DATA_BLOCK "DB00851_St_ConstAiScaleData"   // DB851
TITLE = Static DB [SYSTEM CONSTANTS] — Analog Input Scale Data and Ranges
{ S7_Optimized_Access := 'TRUE' }
AUTHOR : M_Gledhill
FAMILY : SysConstants
NAME : St_ConstAiScaleData
VERSION : 1.0
// PRACTICAL SERIES AUTOMATION LIBRARY (PAL)   —   COPYRIGHT 2020 – M. GLEDHILL (MIT LICENCE)
//                   ———— ◆ ————
// FULL ONLINE DOCUMENTATION IS AVAILABLE AT: https://practicalseries.com/2001-pal/index.html
// stored: AutoNumber false, DBAccessibleFromOPCUA true, IsOnlyStoredInLoadMemory false, IsRetainMemResEnabled false, IsWriteProtectedInAS false, MemoryReserve 100
   VAR
      _DB_Header { ExternalAccessible := 'False'; ExternalVisible := 'False'; ExternalWritable := 'False'} : Array[0..79] of Bool;   // Static DB [SYSTEM CONSTANTS] — Analog Input Scale Data and Ranges
      __________0000_0 { ExternalAccessible := 'False'; ExternalVisible := 'False'; ExternalWritable := 'False'} : Bool := false;
      __________0000_1 { ExternalAccessible := 'False'; ExternalVisible := 'False'; ExternalWritable := 'False'} : Bool := false;
      revInfo { ExternalWritable := 'False'} : "UT01000_St_SysRevision";
      __________0010_0 { ExternalAccessible := 'False'; ExternalVisible := 'False'; ExternalWritable := 'False'} : Bool := false;
      __________0010_1 { ExternalAccessible := 'False'; ExternalVisible := 'False'; ExternalWritable := 'False'} : Bool := false;   // ▀▀▀▀ ANALOG SCALE SIGNALS — TEST SIGNALS
      AI_SCALE_TST001 { ExternalWritable := 'False'; S7_SetPoint := 'True'} : "UT00851_Sy_ConstAiScaleData";   // Test range — 0 to 1000 l/s
      AI_SCALE_TST002 { ExternalWritable := 'False'; S7_SetPoint := 'True'} : "UT00851_Sy_ConstAiScaleData";   // Test range — -500 to +500 l/s
      AI_SCALE_TST003 { ExternalWritable := 'False'; S7_SetPoint := 'True'} : "UT00851_Sy_ConstAiScaleData";   // Test range — -1000 to 0 l/s
      AI_SCALE_TST004 { ExternalWritable := 'False'; S7_SetPoint := 'True'} : "UT00851_Sy_ConstAiScaleData";   // Test range — -270 to +1372 DegC
      AI_SCALE_TST005 { ExternalWritable := 'False'; S7_SetPoint := 'True'} : "UT00851_Sy_ConstAiScaleData";   // Test range — Erroneous configuration
      __________0020_0 { ExternalAccessible := 'False'; ExternalVisible := 'False'; ExternalWritable := 'False'} : Bool := false;
      __________0020_1 { ExternalAccessible := 'False'; ExternalVisible := 'False'; ExternalWritable := 'False'} : Bool := false;   // ▀▀▀▀ ANALOG SCALE SIGNALS — INSTRUMENTS
      AI_SCALE_TST006 { ExternalWritable := 'False'; S7_SetPoint := 'True'} : "UT00851_Sy_ConstAiScaleData";   // Test range — 0 to 1000 l/s
      AI_SCALE_FIC001 { ExternalWritable := 'False'; S7_SetPoint := 'True'} : "UT00851_Sy_ConstAiScaleData";   // Inlet flow meter (0-100 l/s)
      AI_SCALE_LIC001 { ExternalWritable := 'False'; S7_SetPoint := 'True'} : "UT00851_Sy_ConstAiScaleData";   // Inlet tank level (0-50 m3)
      AI_SCALE_PIC301 { ExternalWritable := 'False'; S7_SetPoint := 'True'} : "UT00851_Sy_ConstAiScaleData";   // Inlet filter differential pressure (0-2 BarG)
      AI_SCALE_PIC302 { ExternalWritable := 'False'; S7_SetPoint := 'True'} : "UT00851_Sy_ConstAiScaleData";   // Inlet filter differential pressure (0-2 BarG)
   END_VAR
BEGIN
   // _DB_Header[0] : ▄▄▄▄▄▄▄▄▄▄▄▄▄▄▄▄▄▄▄▄▄▄▄▄▄▄▄▄▄▄▄▄ ＣＯＮＳＴＡＮＴＳ ▄▄
   // _DB_Header[2] : TITLE: SYSTEM CONSTANTS — ANALOG INPUT SCALE DATA AND RANGES
   // _DB_Header[4] : ▀▀▀▀▀▀▀▀▀▀▀▀▀▀▀▀▀▀▀▀▀▀▀▀▀▀▀▀▀▀▀▀▀▀▀▀▀▀▀▀▀▀▀▀
   // _DB_Header[5] : TYPE: STATIC
   // _DB_Header[6] : ▄▄▄▄▄▄▄▄▄▄▄▄▄▄▄▄▄▄▄▄▄▄▄▄▄▄▄▄▄▄▄▄▄▄▄▄▄▄▄▄ ʷᴵᴰ⁻ᵈʰᵇ ▄
   // _DB_Header[8] : DB00851_St_ConstAiScaleData is a static data block that holds a full set of scaled ranges,
   // _DB_Header[9] : engineering units, device tag and descriptive data for all types of analog input scaled signals.
   // _DB_Header[11] : Each dataset is stored in a structure of user data type: UT00851_St_ConstAiScaleData.
   // _DB_Header[12] : This structure is configured to hold all the data required to name, scale and apply engineering
   // _DB_Header[13] : units to an analog input signal.
   // _DB_Header[15] : The scaled signal data is stored as constants and is used by all modules that have an interface
   // _DB_Header[16] : to an analog input card.
   // _DB_Header[18] : The purpose of the user data type and associated data block is to provide a consistent set of
   // _DB_Header[19] : scaled ranges and other data for each device or instrument that is available to the Controller
   // _DB_Header[20] : as an analog input.
   // _DB_Header[22] : The ranges correspond to the scaled values returned by the instrument or device, for example,
   // _DB_Header[23] : a flow meter may have a scaled range of -50 l/s to 200 l/s.
   // _DB_Header[25] : In addition, each dataset contains the instrument or device tag (e.g. FIC001), the engineering
   // _DB_Header[26] : units in use (e.g. l/s, kg/hour, °C, % &c.), over-range and under-range limits, a textual description
   // _DB_Header[27] : of the function of the instrument or device e.g. inlet flowmeter (0 l/s to 100 l/s) and additional
   // _DB_Header[28] : user specific information.
   // _DB_Header[30] : The PDF version of the SMDS for this module is available online here:
   // _DB_Header[31] : http://psop.uk/pal-smds-db00851-p
   // _DB_Header[33] : ━━━ ⬙⬙⬙⬙⬙⬙ ━━━
   // _DB_Header[35] : ▄▄▄▄▄▄▄▄▄▄▄▄▄▄▄▄▄▄▄▄▄▄▄▄▄▄▄▄▄▄▄▄▄▄▄▄▄▄▄▄▄▄▄▄
   // _DB_Header[36] : MODIFICATION HISTORY
   // _DB_Header[38] : This is a summary of the recent software modifications made to this block (most recent at top)
   // _DB_Header[40] : ―――――――――――――――――――――――――――――――――――――――――――
   // _DB_Header[41] : DATE REVISION MASTER BRANCH DEV
   // _DB_Header[42] : (nnn.amm) COMMIT TAG (Base ---> Merge) BRANCH Author
   // _DB_Header[43] : ———————————————————————————————————————————
   // _DB_Header[44] : 2022.05.15 001.000 D0018 D0017 D0018 None M. Gledhill
   // _DB_Header[45] : DB00851 — RELEASED FOR USE
   // _DB_Header[46] : Merge back to master branch
   // _DB_Header[48] : 2024.05.15 001.000 D0017A-000.104 D0017 N/A D0017A M. Gledhill
   // _DB_Header[49] : DB00851 — RELEASED FOR USE
   // _DB_Header[51] : 2024.05.03 000.801 D0017A-000.102 D0017 N/A D0017A M. Gledhill
   // _DB_Header[52] : DB00851 Block populated
   // _DB_Header[54] : 2024.04.09 000.101 D0017A-000.101 D0017 N/A D0017A M. Gledhill
   // _DB_Header[55] : DB00851 Block created
   // _DB_Header[56] : ———————————————————————————————————————————
   // _DB_Header[57] : Where: nnn = Major revision
   // _DB_Header[58] : a = Type (1-7 Development, 8 Proving, 9 Qualification, 0 Release)
   // _DB_Header[59] : mm = Minor revision (must be 00 if a = 0)
   // _DB_Header[60] : Block properties version number should be set to nn.a (only one decimal place)
   // _DB_Header[62] : ██████████████ █ █ █ █ END █ █ █ █ ██████████████
   revInfo.REV_BLOCK := 'DB00851';
   revInfo.REV_NUMBER := '001.000';
   revInfo.REV_DATE := '2024-05-15';
   revInfo.REV_AUTHOR := 'M. Gledhill';
   AI_SCALE_TST001.AI_TAG := 'TST001';
   AI_SCALE_TST001.SCALE_MIN := 0.0;
   AI_SCALE_TST001.SCALE_MAX := 1000.0;
   AI_SCALE_TST001.SCALE_UNITS := 'l/s';
   AI_SCALE_TST001.SCALE_DESC := 'Test Range (0 to 1000 l/s)';
   AI_SCALE_TST001.LIMIT_UNDER := -62.5;
   AI_SCALE_TST001.LIMIT_OVER := 1062.5;
   AI_SCALE_TST002.AI_TAG := 'TST002';
   AI_SCALE_TST002.SCALE_MIN := -500.0;
   AI_SCALE_TST002.SCALE_MAX := 500.0;
   AI_SCALE_TST002.SCALE_UNITS := 'l/s';
   AI_SCALE_TST002.SCALE_DESC := 'Test Range (-500 to 500 l/s)';
   AI_SCALE_TST002.LIMIT_UNDER := -562.5;
   AI_SCALE_TST002.LIMIT_OVER := 562.5;
   AI_SCALE_TST003.AI_TAG := 'TST003';
   AI_SCALE_TST003.SCALE_MIN := -1000.0;
   AI_SCALE_TST003.SCALE_MAX := 0.0;
   AI_SCALE_TST003.SCALE_UNITS := 'l/s';
   AI_SCALE_TST003.SCALE_DESC := 'Test Range (-1000 to 0 l/s)';
   AI_SCALE_TST003.LIMIT_UNDER := -1062.5;
   AI_SCALE_TST003.LIMIT_OVER := 62.5;
   AI_SCALE_TST004.AI_TAG := 'TST005';
   AI_SCALE_TST004.SCALE_MIN := -270.0;
   AI_SCALE_TST004.SCALE_MAX := 1372.0;
   AI_SCALE_TST004.SCALE_UNITS := 'DegC';
   AI_SCALE_TST004.SCALE_DESC := 'Test Range (-270 to +1372 DegC)';
   AI_SCALE_TST004.LIMIT_UNDER := -300.0;
   AI_SCALE_TST004.LIMIT_OVER := 1400.0;
   AI_SCALE_TST005.AI_TAG := 'TST005';
   AI_SCALE_TST005.___________0020_0 := false;
   AI_SCALE_TST005.___________0020_1 := false;
   AI_SCALE_TST005.SCALE_MIN := 0.0;
   AI_SCALE_TST005.SCALE_MAX := 1000.0;
   AI_SCALE_TST005.SCALE_UNITS := 'l/s';
   AI_SCALE_TST005.SCALE_DESC := 'Test Range (0 to 1000 l/s)';
   AI_SCALE_TST005.___________0030_0 := false;
   AI_SCALE_TST005.___________0030_1 := false;
   AI_SCALE_TST005.LIMIT_UNDER := 100.0;
   AI_SCALE_TST005.LIMIT_OVER := 900.0;
   AI_SCALE_TST006.AI_TAG := 'TST005';
   AI_SCALE_TST006.SCALE_MIN := 0.0;
   AI_SCALE_TST006.SCALE_MAX := 1000.0;
   AI_SCALE_TST006.SCALE_UNITS := 'l/s';
   AI_SCALE_TST006.SCALE_DESC := 'Test Range (0 to 1000 l/s)';
   AI_SCALE_TST006.LIMIT_UNDER := 100.0;
   AI_SCALE_TST006.LIMIT_OVER := 900.0;
   AI_SCALE_FIC001.AI_TAG := 'FIC001';
   AI_SCALE_FIC001.SCALE_MIN := 0.0;
   AI_SCALE_FIC001.SCALE_MAX := 100.0;
   AI_SCALE_FIC001.SCALE_UNITS := 'l/s';
   AI_SCALE_FIC001.SCALE_DESC := 'Inlet flow meter (0-100 l/s)';
   AI_SCALE_FIC001.LIMIT_UNDER := -5.0;
   AI_SCALE_FIC001.LIMIT_OVER := 105.0;
   AI_SCALE_FIC001.USER_INFO_1 := 'Instrument manufacturer: Siemens';
   AI_SCALE_FIC001.USER_INFO_2 := 'Instrument type: Sitrans FM MAG 5000 (mass flow)';
   AI_SCALE_FIC001.USER_INFO_3 := 'Instrument part no.: 7ME5920-1AA10-1AA0';
   AI_SCALE_FIC001.USER_INFO_4 := 'Instrument serial no.: 3443201102';
   AI_SCALE_LIC001.AI_TAG := 'LIC001';
   AI_SCALE_LIC001.SCALE_MIN := 0.0;
   AI_SCALE_LIC001.SCALE_MAX := 50.0;
   AI_SCALE_LIC001.SCALE_UNITS := 'm3';
   AI_SCALE_LIC001.SCALE_DESC := 'Inlet tank level (0-50 m3)';
   AI_SCALE_LIC001.LIMIT_UNDER := -2.5;
   AI_SCALE_LIC001.LIMIT_OVER := 52.5;
   AI_SCALE_LIC001.USER_INFO_1 := 'Instrument manufacturer: Siemens';
   AI_SCALE_LIC001.USER_INFO_2 := 'Instrument type: Sitrans LU240 (level)';
   AI_SCALE_LIC001.USER_INFO_3 := 'Instrument part no.: 7ML5110-1DD07-4AF0';
   AI_SCALE_LIC001.USER_INFO_4 := 'Instrument serial no.: 4514461005';
   AI_SCALE_PIC301.AI_TAG := 'PIC301';
   AI_SCALE_PIC301.SCALE_MIN := 0.0;
   AI_SCALE_PIC301.SCALE_MAX := 2.0;
   AI_SCALE_PIC301.SCALE_UNITS := 'BarG';
   AI_SCALE_PIC301.SCALE_DESC := 'Inlet filter differential pressure (0-2 BarG)';
   AI_SCALE_PIC301.LIMIT_UNDER := -0.1;
   AI_SCALE_PIC301.LIMIT_OVER := 2.1;
   AI_SCALE_PIC301.USER_INFO_1 := 'Instrument manufacturer: Siemens';
   AI_SCALE_PIC301.USER_INFO_2 := 'Instrument type: Sitrans P420 (pressure)';
   AI_SCALE_PIC301.USER_INFO_3 := 'Instrument part no.: 7MF0440-1ML02-5BF0';
   AI_SCALE_PIC301.USER_INFO_4 := 'Instrument serial no.: 7875344001';
   AI_SCALE_PIC302.AI_TAG := 'PIC301';
   AI_SCALE_PIC302.SCALE_MIN := 0.0;
   AI_SCALE_PIC302.SCALE_MAX := 2.0;
   AI_SCALE_PIC302.SCALE_UNITS := 'BarG';
   AI_SCALE_PIC302.SCALE_DESC := 'Inlet filter differential pressure (0-2 BarG)';
   AI_SCALE_PIC302.LIMIT_UNDER := -0.1;
   AI_SCALE_PIC302.LIMIT_OVER := 2.1;
   AI_SCALE_PIC302.USER_INFO_1 := 'Instrument manufacturer: Siemens';
   AI_SCALE_PIC302.USER_INFO_2 := 'Instrument type: Sitrans P420 (pressure)';
   AI_SCALE_PIC302.USER_INFO_3 := 'Instrument part no.: 7MF0440-1ML02-5BF0';
   AI_SCALE_PIC302.USER_INFO_4 := 'Instrument serial no.: 7875344008';
END_DATA_BLOCK

DATA_BLOCK "DB00852_St_ConstAqScaleData"   // DB852
TITLE = Static DB [SYSTEM CONSTANTS] — Analog Input Scale Data and Ranges
{ S7_Optimized_Access := 'TRUE' }
AUTHOR : M_Gledhill
FAMILY : SysConstants
NAME : St_ConstAiScaleData
VERSION : 1.0
// PRACTICAL SERIES AUTOMATION LIBRARY (PAL)   —   COPYRIGHT 2020 – M. GLEDHILL (MIT LICENCE)
//                   ———— ◆ ————
// FULL ONLINE DOCUMENTATION IS AVAILABLE AT: https://practicalseries.com/2001-pal/index.html
// stored: AutoNumber false, DBAccessibleFromOPCUA true, IsOnlyStoredInLoadMemory false, IsRetainMemResEnabled false, IsWriteProtectedInAS false, MemoryReserve 100
   VAR
      _DB_Header { ExternalAccessible := 'False'; ExternalVisible := 'False'; ExternalWritable := 'False'} : Array[0..79] of Bool;   // Static DB [SYSTEM CONSTANTS] — Analog Instrument Scale Data and Ranges
      __________0000_0 { ExternalAccessible := 'False'; ExternalVisible := 'False'; ExternalWritable := 'False'} : Bool := false;
      __________0000_1 { ExternalAccessible := 'False'; ExternalVisible := 'False'; ExternalWritable := 'False'} : Bool := false;
      revInfo { ExternalWritable := 'False'} : "UT01000_St_SysRevision";
      __________0010_0 { ExternalAccessible := 'False'; ExternalVisible := 'False'; ExternalWritable := 'False'} : Bool := false;
      __________0010_1 { ExternalAccessible := 'False'; ExternalVisible := 'False'; ExternalWritable := 'False'} : Bool := false;   // ▀▀▀▀ ANALOG SCALE SIGNALS — MODULATING VALVES
      AQ_SCALE_FCV001_DMD { ExternalWritable := 'False'; S7_SetPoint := 'True'} : "UT00852_Sy_ConstAqScaleData";   // Inlet flow control valve position demand (0 to 100%)
      __________0020_0 { ExternalAccessible := 'False'; ExternalVisible := 'False'; ExternalWritable := 'False'} : Bool := false;
      __________0020_1 { ExternalAccessible := 'False'; ExternalVisible := 'False'; ExternalWritable := 'False'} : Bool := false;   // ▀▀▀▀ ANALOG SCALE SIGNALS — CHART RECORDER
      AQ_SCALE_REC001 { ExternalWritable := 'False'; S7_SetPoint := 'True'} : "UT00852_Sy_ConstAqScaleData";   // Recorder - Inlet flow meter (0-100 l/s)
      AQ_SCALE_REC002 { ExternalWritable := 'False'; S7_SetPoint := 'True'} : "UT00852_Sy_ConstAqScaleData";   // Recorder - Inlet tank level (0-50 m3)
   END_VAR
BEGIN
   // _DB_Header[0] : ▄▄▄▄▄▄▄▄▄▄▄▄▄▄▄▄▄▄▄▄▄▄▄▄▄▄▄▄▄▄▄▄ ＣＯＮＳＴＡＮＴＳ ▄▄
   // _DB_Header[2] : TITLE: SYSTEM CONSTANTS — ANALOG INPUT SCALE DATA AND RANGES
   // _DB_Header[4] : ▀▀▀▀▀▀▀▀▀▀▀▀▀▀▀▀▀▀▀▀▀▀▀▀▀▀▀▀▀▀▀▀▀▀▀▀▀▀▀▀▀▀▀▀
   // _DB_Header[5] : TYPE: STATIC
   // _DB_Header[6] : ▄▄▄▄▄▄▄▄▄▄▄▄▄▄▄▄▄▄▄▄▄▄▄▄▄▄▄▄▄▄▄▄▄▄▄▄▄▄▄▄ ʷᴵᴰ⁻ᵈʰᵇ ▄
   // _DB_Header[8] : DB00852_St_ConstAqScaleData is a static data block that holds a full set of scaled ranges,
   // _DB_Header[9] : engineering units, device tag and descriptive data for all types of analog output scaled signals.
   // _DB_Header[11] : Each dataset is stored in a structure of user data type: UT00852_St_ConstAqScaleData.
   // _DB_Header[12] : This structure is configured to hold all the data required to name, scale and apply engineering
   // _DB_Header[13] : units to an analog output signal.
   // _DB_Header[15] : All the scaled signal data is stored as constants and is used by all modules that have an interface
   // _DB_Header[16] : to an analog output card.
   // _DB_Header[18] : The purpose of the user data type and associated data block is to provide a consistent set of
   // _DB_Header[19] : scaled ranges and other data for each device that is available to the Controller
   // _DB_Header[20] : as an analog output.
   // _DB_Header[22] : The ranges correspond to the scaled values of a signal that is to be converted into an analog
   // _DB_Header[23] : output, for example, a modulating valve may have a scaled range of 0% to 100%.
   // _DB_Header[25] : In addition, each dataset contains the device tag (e.g. FCV001), the engineering
   // _DB_Header[26] : units in use (e.g. l/s, kg/hour, °C, % &c.), over-range and under-range limits, a textual description
   // _DB_Header[27] : of the function of the device e.g.inlet flow control valve and additional user specific
   // _DB_Header[28] : information.
   // _DB_Header[30] : The PDF version of the SMDS for this module is available online here:
   // _DB_Header[31] : http://psop.uk/pal-smds-db00851-p
   // _DB_Header[33] : ━━━ ⬙⬙⬙⬙⬙⬙ ━━━
   // _DB_Header[35] : ▄▄▄▄▄▄▄▄▄▄▄▄▄▄▄▄▄▄▄▄▄▄▄▄▄▄▄▄▄▄▄▄▄▄▄▄▄▄▄▄▄▄▄▄
   // _DB_Header[36] : MODIFICATION HISTORY
   // _DB_Header[38] : This is a summary of the recent software modifications made to this block (most recent at top)
   // _DB_Header[40] : ―――――――――――――――――――――――――――――――――――――――――――
   // _DB_Header[41] : DATE REVISION MASTER BRANCH DEV
   // _DB_Header[42] : (nnn.amm) COMMIT TAG (Base ---> Merge) BRANCH Author
   // _DB_Header[43] : ———————————————————————————————————————————
   // _DB_Header[44] : 2024.05.17 001.000 D0017A-000.104 D0017 N/A D0017A M. Gledhill
   // _DB_Header[45] : DB00852 — RELEASED FOR USE
   // _DB_Header[47] : 2024.05.03 000.801 D0017A-000.102 D0017 N/A D0017A M. Gledhill
   // _DB_Header[48] : DB00852 Block populated
   // _DB_Header[50] : 2024.04.09 000.101 D0017A-000.101 D0017 N/A D0017A M. Gledhill
   // _DB_Header[51] : DB00852 Block created
   // _DB_Header[52] : ———————————————————————————————————————————
   // _DB_Header[53] : Where: nnn = Major revision
   // _DB_Header[54] : a = Type (1-7 Development, 8 Proving, 9 Qualification, 0 Release)
   // _DB_Header[55] : mm = Minor revision (must be 00 if a = 0)
   // _DB_Header[56] : Block properties version number should be set to nn.a (only one decimal place)
   // _DB_Header[58] : ██████████████ █ █ █ █ END █ █ █ █ ██████████████
   revInfo.REV_BLOCK := 'DB00852';
   revInfo.REV_NUMBER := '001.000';
   revInfo.REV_DATE := '2024-05-17';
   revInfo.REV_AUTHOR := 'M. Gledhill';
   AQ_SCALE_FCV001_DMD.AQ_TAG := 'FCV001';
   AQ_SCALE_FCV001_DMD.SCALE_MIN := 0.0;
   AQ_SCALE_FCV001_DMD.SCALE_MAX := 100.0;
   AQ_SCALE_FCV001_DMD.SCALE_UNITS := '%';
   AQ_SCALE_FCV001_DMD.SCALE_DESC := 'Inlet flow control valve (0 to 100%)';
   AQ_SCALE_FCV001_DMD.LIMIT_UNDER := -2.5;
   AQ_SCALE_FCV001_DMD.LIMIT_OVER := 102.5;
   AQ_SCALE_FCV001_DMD.USER_INFO_1 := 'Instrument manufacturer: Siemens';
   AQ_SCALE_FCV001_DMD.USER_INFO_2 := 'Instrument type: 2-port magnetic';
   AQ_SCALE_FCV001_DMD.USER_INFO_3 := 'Instrument part no.: MXG461.15-0.6';
   AQ_SCALE_FCV001_DMD.USER_INFO_4 := 'Instrument serial no.:2075181118';
   AQ_SCALE_REC001.AQ_TAG := 'REC001';
   AQ_SCALE_REC001.SCALE_MIN := 0.0;
   AQ_SCALE_REC001.SCALE_MAX := 100.0;
   AQ_SCALE_REC001.SCALE_UNITS := 'l/s';
   AQ_SCALE_REC001.SCALE_DESC := 'Recorder - Inlet flow meter (0-100 l/s)';
   AQ_SCALE_REC002.AQ_TAG := 'REC002';
   AQ_SCALE_REC002.SCALE_MIN := 0.0;
   AQ_SCALE_REC002.SCALE_MAX := 50.0;
   AQ_SCALE_REC002.SCALE_UNITS := 'm3';
   AQ_SCALE_REC002.SCALE_DESC := 'Recorder - Inlet tank level (0-50 m3)';
END_DATA_BLOCK

DATA_BLOCK "DB21001_Dy_SysGlobalData"   // DB21001
TITLE = Dynamic DB — Sys - Global Data
{ S7_Optimized_Access := 'TRUE' }
AUTHOR : M_Gledhill
FAMILY : System
NAME : Dy_SysGlobalData
VERSION : 1.0
// PRACTICAL SERIES AUTOMATION LIBRARY (PAL)   —   COPYRIGHT 2020 – M. GLEDHILL (MIT LICENCE)
//                   ———— ◆ ————
//  FOR DETAILED DOCUMENTATION — SELECT THE BLOCK IN THE PROJECT TREE AND PRESS SHIFT + F1
//  FULL ONLINE DOCUMENTATION IS AVAILABLE AT: https://practicalseries.com/2001-pal/index.html
// stored: AutoNumber false, DBAccessibleFromOPCUA true, IsOnlyStoredInLoadMemory false, IsRetainMemResEnabled false, IsWriteProtectedInAS false, MemoryReserve 100
   VAR
      _DB_Header { ExternalWritable := 'False'} : Array[0..79] of Bool;   // STANDARD SYSTEM GLOBAL DATA
      __________0000_0 { ExternalWritable := 'False'} : Bool := false;
      __________0000_1 { ExternalWritable := 'False'} : Bool := false;   // ▀▀▀▀ DB CURRENT REVISION
      revInfo { ExternalWritable := 'False'} : "UT01000_St_SysRevision";
      __________0010_0 { ExternalWritable := 'False'} : Bool := false;
      __________0010_1 { ExternalWritable := 'False'} : Bool := false;   // ▀▀▀▀ PROJECT CURRENT REVISION
      projRevInfo { ExternalWritable := 'False'} : "UT01000_St_SysRevision";
      __________0020_0 { ExternalWritable := 'False'} : Bool := false;
      __________0020_1 { ExternalWritable := 'False'} : Bool := false;   // ▀▀▀▀ SYSTEM SIGNALS — LOGIC AND TIMING SIGNALS
      SysSignals { ExternalWritable := 'False'} : "UT21000_Dy_SysSignals";
      __________0030_0 { ExternalWritable := 'False'} : Bool := false;
      __________0030_1 { ExternalWritable := 'False'} : Bool := false;   // ▀▀▀▀ SYSTEM DATA — CYCLE TIMING AND RTC
      SysData { ExternalWritable := 'False'} : "UT21001_Dy_SysData";
      __________0040_0 { ExternalWritable := 'False'} : Bool := false;
      __________0040_1 { ExternalWritable := 'False'} : Bool := false;   // ▀▀▀▀ OB CALL TIMES
      OB10_CallTime { ExternalWritable := 'False'} : DTL;   // Time of day interrupt 1
      OB11_CallTime { ExternalWritable := 'False'} : DTL;   // Time of day interrupt 2
      OB12_CallTime { ExternalWritable := 'False'} : DTL;   // Time of day interrupt 3
      OB13_CallTime { ExternalWritable := 'False'} : DTL;   // Time of day interrupt 4
      OB14_CallTime { ExternalWritable := 'False'} : DTL;   // Time of day interrupt 5
      OB15_CallTime { ExternalWritable := 'False'} : DTL;   // Time of day interrupt 6
      OB16_CallTime { ExternalWritable := 'False'} : DTL;   // Time of day interrupt 7
      OB17_CallTime { ExternalWritable := 'False'} : DTL;   // Time of day interrupt 8
      OB20_CallTime { ExternalWritable := 'False'} : DTL;   // Time delay interrupt 1
      OB21_CallTime { ExternalWritable := 'False'} : DTL;   // Time delay interrupt 2
      OB22_CallTime { ExternalWritable := 'False'} : DTL;   // Time delay interrupt 3
      OB23_CallTime { ExternalWritable := 'False'} : DTL;   // Time delay interrupt 4
      OB30_CallTime { ExternalWritable := 'False'} : DTL;   // Timed cyclic interrupt 1
      OB31_CallTime { ExternalWritable := 'False'} : DTL;   // Timed cyclic interrupt 2
      OB32_CallTime { ExternalWritable := 'False'} : DTL;   // Timed cyclic interrupt 3
      OB33_CallTime { ExternalWritable := 'False'} : DTL;   // Timed cyclic interrupt 4
      OB34_CallTime { ExternalWritable := 'False'} : DTL;   // Timed cyclic interrupt 5
      OB35_CallTime { ExternalWritable := 'False'} : DTL;   // Timed cyclic interrupt 6
      OB36_CallTime { ExternalWritable := 'False'} : DTL;   // Timed cyclic interrupt 7
      OB37_CallTime { ExternalWritable := 'False'} : DTL;   // Timed cyclic interrupt 8
      OB38_CallTime { ExternalWritable := 'False'} : DTL;   // Timed cyclic interrupt 9
      OB40_CallTime { ExternalWritable := 'False'} : DTL;   // Hardware interrupt 1
      OB41_CallTime { ExternalWritable := 'False'} : DTL;   // Hardware interrupt 2
      OB42_CallTime { ExternalWritable := 'False'} : DTL;   // Hardware interrupt 3
      OB43_CallTime { ExternalWritable := 'False'} : DTL;   // Hardware interrupt 4
      OB44_CallTime { ExternalWritable := 'False'} : DTL;   // Hardware interrupt 5
      OB45_CallTime { ExternalWritable := 'False'} : DTL;   // Hardware interrupt 6
      OB46_CallTime { ExternalWritable := 'False'} : DTL;   // Hardware interrupt 7
      OB47_CallTime { ExternalWritable := 'False'} : DTL;   // Hardware interrupt 8
      OB80_CallTime { ExternalWritable := 'False'} : DTL;   // Error interrupt — max cycle time exceeded
      OB82_CallTime { ExternalWritable := 'False'} : DTL;   // Error interrupt — module diagnostic
      OB83_CallTime { ExternalWritable := 'False'} : DTL;   // Error interrupt — module changed
      OB86_CallTime { ExternalWritable := 'False'} : DTL;   // Error interrupt — rack fault
      OB100_CallTime { ExternalWritable := 'False'} : DTL;   // Start-up interrupt
      OB121_CallTime { ExternalWritable := 'False'} : DTL;   // Error interrupt — programming fault
      OB122_CallTime { ExternalWritable := 'False'} : DTL;   // Error interrupt — IO access fault
   END_VAR
BEGIN
   // _DB_Header[0] : ▀▀▀▀▀▀▀▀▀▀▀▀▀▀▀▀▀▀▀▀▀▀▀▀▀▀▀▀▀▀▀▀▀▀▀▀▀▀▀▀▀▀▀▀
   // _DB_Header[2] : TITLE: STANDARD SYSTEM GLOBAL DATA
   // _DB_Header[4] : ▄▄▄▄▄▄▄▄▄▄▄▄▄▄▄▄▄▄▄▄▄▄▄▄▄▄▄▄▄▄▄▄▄▄▄▄▄▄▄▄▄▄▄▄
   // _DB_Header[5] : TYPE: DYNAMIC
   // _DB_Header[6] : ▀▀▀▀▀▀▀▀▀▀▀▀▀▀▀▀▀▀▀▀▀▀▀▀▀▀▀▀▀▀▀▀▀▀▀▀▀▀▀▀▀▀▀▀
   // _DB_Header[8] : Global system data storage DB. The block records various system variables and information:
   // _DB_Header[10] : • Project revision data
   // _DB_Header[11] : • Common system signals (logic and timing)
   // _DB_Header[12] : • Cycle timing information (previous, max, min and a cycle counter)
   // _DB_Header[13] : • CPU real time clock data (in globally readable format)
   // _DB_Header[14] : • Last call time of any interrupt OB
   // _DB_Header[16] : The cycle timing information and the RTC data are provided by FC01000. The interrupt OB data
   // _DB_Header[17] : is provided by the individual OBs.
   // _DB_Header[19] : ━━━ ⬙⬙⬙⬙⬙⬙ ━━━
   // _DB_Header[21] : ▄▄▄▄▄▄▄▄▄▄▄▄▄▄▄▄▄▄▄▄▄▄▄▄▄▄▄▄▄▄▄▄▄▄▄▄▄▄▄▄▄▄▄▄
   // _DB_Header[22] : MODIFICATION HISTORY
   // _DB_Header[24] : This is a summary of the recent software modifications made to this block (most recent at top)
   // _DB_Header[26] : ―――――――――――――――――――――――――――――――――――――――――――
   // _DB_Header[27] : DATE REVISION MASTER BRANCH DEV
   // _DB_Header[28] : (nnn.amm) COMMIT TAG (Base ---> Merge) BRANCH Author
   // _DB_Header[29] : ———————————————————————————————————————————
   // _DB_Header[30] : 2021.05.11 001.000 D0006 D0005 D0006 None M. Gledhill
   // _DB_Header[31] : FC01001 — RELEASED FOR USE
   // _DB_Header[32] : Merge back to master branch
   // _DB_Header[34] : 2021.05.11 000.801 D0005A-000.801 D0005 N/A D0005A M. Gledhill
   // _DB_Header[35] : FC01001 — Released for SMT
   // _DB_Header[37] : 2021.05.08 000.101 D0005A-000.101 D0005 N/A D0005A M. Gledhill
   // _DB_Header[38] : FC01001 Migration to VCS
   // _DB_Header[39] : ———————————————————————————————————————————
   // _DB_Header[41] : ██████████████ █ █ █ █ END █ █ █ █ ██████████████
   revInfo.REV_BLOCK := 'DB21001';
   revInfo.REV_NUMBER := '001.000';
   revInfo.REV_DATE := '2021-05-11';
   revInfo.REV_AUTHOR := 'M. Gledhill';
END_DATA_BLOCK

DATA_BLOCK "DB02001_St_InstAnalogRead"   // DB2001
TITLE = Static DB — Inst - Analog Instrument Read, Scale and Monitor
{ S7_Optimized_Access := 'TRUE' }
AUTHOR : M_Gledhill
FAMILY : Instrumentation
NAME : St_InstAnalogRead
VERSION : 0.1
// PRACTICAL SERIES AUTOMATION LIBRARY (PAL)   —   COPYRIGHT 2020 – M. GLEDHILL (MIT LICENCE)
//                   ———— ◆ ————
//  FOR DETAILED DOCUMENTATION — SELECT THE BLOCK IN THE PROJECT TREE AND PRESS SHIFT + F1
//  FULL ONLINE DOCUMENTATION IS AVAILABLE AT: https://practicalseries.com/2001-pal/index.html
// stored: AutoNumber false, DBAccessibleFromOPCUA true, IsOnlyStoredInLoadMemory false, IsRetainMemResEnabled false, IsWriteProtectedInAS false, MemoryReserve 100
   VAR
      _DB_Header { ExternalAccessible := 'False'; ExternalVisible := 'False'; ExternalWritable := 'False'} : Array[0..79] of Bool;   // STANDARD ANALOG INSTRUMENT READ
      __________0000_0 { ExternalAccessible := 'False'; ExternalVisible := 'False'; ExternalWritable := 'False'} : Bool := false;
      __________0000_1 { ExternalAccessible := 'False'; ExternalVisible := 'False'; ExternalWritable := 'False'} : Bool := false;   // ▀▀▀▀ DB CURRENT REVISION
      revInfo { ExternalWritable := 'False'; S7_SetPoint := 'True'} : "UT01000_St_SysRevision";
      __________0010_0 { ExternalAccessible := 'False'; ExternalVisible := 'False'; ExternalWritable := 'False'} : Bool := false;
      __________0010_1 { ExternalAccessible := 'False'; ExternalVisible := 'False'; ExternalWritable := 'False'} : Bool := false;   // ▀▀▀▀ ANALOG INSTRUMENTS
      FIC101 { ExternalWritable := 'False'; S7_SetPoint := 'True'} : "UT02001_St_InstAnalogRead";   // Filter 1 outlet flow
   END_VAR
BEGIN
   // _DB_Header[0] : ▀▀▀▀▀▀▀▀▀▀▀▀▀▀▀▀▀▀▀▀▀▀▀▀▀▀▀▀▀▀▀▀▀▀▀▀▀▀▀▀▀▀▀▀
   // _DB_Header[2] : TITLE: STANDARD ANALOG INSTRUMENT READ (SCALE & ALARM MONITORING)
   // _DB_Header[4] : ▄▄▄▄▄▄▄▄▄▄▄▄▄▄▄▄▄▄▄▄▄▄▄▄▄▄▄▄▄▄▄▄▄▄▄▄▄▄▄▄▄▄▄▄
   // _DB_Header[5] : TYPE: STATIC
   // _DB_Header[6] : ▀▀▀▀▀▀▀▀▀▀▀▀▀▀▀▀▀▀▀▀▀▀▀▀▀▀▀▀▀▀▀▀▀▀▀▀▀▀▀▀▀▀▀▀
   // _DB_Header[8] : This is the static data block associated with the standard analog instrument read
   // _DB_Header[9] : block:
   // _DB_Header[10] : FC02001_StdInstAnalogRead
   // _DB_Header[12] : The static data holds the threshold values for any configured alarms and warnings,
   // _DB_Header[13] : activation delays, scaled and raw value ranges and various configuration options.
   // _DB_Header[15] : Each instrument is given the user data type:
   // _DB_Header[16] : UT02001_St_InstAnalogRead
   // _DB_Header[17] : This holds the full set of static configuration data for the instrument.
   // _DB_Header[19] : ━━━ ⬙⬙⬙⬙⬙⬙ ━━━
   // _DB_Header[21] : ▄▄▄▄▄▄▄▄▄▄▄▄▄▄▄▄▄▄▄▄▄▄▄▄▄▄▄▄▄▄▄▄▄▄▄▄▄▄▄▄▄▄▄▄
   // _DB_Header[22] : MODIFICATION HISTORY
   // _DB_Header[24] : This is a summary of the recent software modifications made to this block (most recent at top)
   // _DB_Header[26] : ―――――――――――――――――――――――――――――――――――――――――――
   // _DB_Header[27] : DATE REVISION MASTER BRANCH DEV
   // _DB_Header[28] : (nnn.amm) COMMIT TAG (Base ---> Merge) BRANCH Author
   // _DB_Header[29] : ———————————————————————————————————————————
   // _DB_Header[30] : 2021.05.18 000.101 D0006B-000.101 D0006 N/A D0006B M. Gledhill
   // _DB_Header[31] : FC02001 Migration to VCS
   // _DB_Header[32] : ———————————————————————————————————————————
   // _DB_Header[33] : Where: nnn = Major revision
   // _DB_Header[34] : a = Type (1-7 Development, 8 Proving, 9 Qualification, 0 Release)
   // _DB_Header[35] : mm = Minor revision (must be 00 if a = 0)
   // _DB_Header[36] : Block properties version number should be set to nn.a (only one decimal place)
   // _DB_Header[38] : ██████████████ █ █ █ █ END █ █ █ █ ██████████████
   revInfo.REV_BLOCK := 'DB02001';
   revInfo.REV_NUMBER := '000.101';
   revInfo.REV_DATE := '2021-05-18';
   revInfo.REV_AUTHOR := 'M. Gledhill';
   FIC101.CONFIG_ALM_H_ENABLE := true;
   FIC101.CONFIG_ALM_L_ENABLE := true;
   FIC101.CONFIG_WRN_H_ENABLE := true;
   FIC101.CONFIG_WRN_L_ENABLE := true;
   FIC101.CONFIG_FP_DISABLE := false;
   FIC101.CONFIG_SIM_DISABLE := false;
   FIC101.CONFIG_RL_ENABLE := false;
   FIC101.RANGE_RAW_MAX := 27648;
   FIC101.RANGE_SCALE_MIN := 0.0;
   FIC101.RANGE_SCALE_MAX := 1000.0;
   FIC101.RANGE_OOR_PERCENT := 2.5;
   FIC101.INFO_TAG := 'FIC101';
   FIC101.INFO_UNITS := 'l/s';
   FIC101.SP_ALM_H_VAL := 750.0;
   FIC101.SP_ALM_L_VAL := 250.0;
   FIC101.SP_WRN_H_VAL := 625.0;
   FIC101.SP_WRN_L_VAL := 375.0;
   FIC101.SP_ALM_H_HYST_VAL := 62.5;
   FIC101.SP_ALM_L_HYST_VAL := 62.0;
   FIC101.SP_WRN_H_HYST_VAL := 61.5;
   FIC101.SP_WRN_L_HYST_VAL := 61.0;
   FIC101.TIME_ALM_H_ON_DEL := 10.0;
   FIC101.TIME_ALM_L_ON_DEL := 11.0;
   FIC101.TIME_WRN_H_ON_DEL := 12.0;
   FIC101.TIME_WRN_L_ON_DEL := 13.0;
   FIC101.TIME_ALM_H_OFF_DEL := 15.0;
   FIC101.TIME_ALM_L_OFF_DEL := 16.0;
   FIC101.TIME_WRN_H_OFF_DEL := 17.0;
   FIC101.TIME_WRN_L_OFF_DEL := 18.0;
END_DATA_BLOCK

DATA_BLOCK "DB22001_Dy_InstAnalogRead"   // DB22001
TITLE = Dynamic DB [INSTRUMENTATION] — Analog Instrument Read, Scale and Monitor
{ S7_Optimized_Access := 'TRUE' }
AUTHOR : M_Gledhill
FAMILY : Instrumentation
NAME : Dy_InstAnalogRead
VERSION : 3.0
// PRACTICAL SERIES AUTOMATION LIBRARY (PAL)   —   COPYRIGHT 2020 – M. GLEDHILL (MIT LICENCE)
//                   ———— ◆ ————
// FULL ONLINE DOCUMENTATION IS AVAILABLE AT: https://practicalseries.com/2001-pal/index.html
// stored: AutoNumber false, DBAccessibleFromOPCUA true, IsOnlyStoredInLoadMemory false, IsRetainMemResEnabled false, IsWriteProtectedInAS false, MemoryReserve 100
   VAR
      _DB_Header { ExternalAccessible := 'False'; ExternalVisible := 'False'; ExternalWritable := 'False'} : Array[0..79] of Bool;   // Dynamic DB [INSTRUMENTATION] — Analog Instrument Read, Scale and Monitor
      __________0000_0 { ExternalAccessible := 'False'; ExternalVisible := 'False'; ExternalWritable := 'False'} : Bool := false;
      __________0000_1 { ExternalAccessible := 'False'; ExternalVisible := 'False'; ExternalWritable := 'False'} : Bool := false;   // ▀▀▀▀ DB CURRENT REVISION
      revInfo { ExternalWritable := 'False'; S7_SetPoint := 'True'} : "UT01000_St_SysRevision";   // Revision information
      __________0010_0 { ExternalAccessible := 'False'; ExternalVisible := 'False'; ExternalWritable := 'False'} : Bool := false;
      __________0010_1 { ExternalAccessible := 'False'; ExternalVisible := 'False'; ExternalWritable := 'False'} : Bool := false;   // ▀▀▀▀ ANALOG INSTRUMENTS
      FIC101 { S7_SetPoint := 'True'} : "UT22001_Dy_InstAnalogRead";   // Filter 1 outlet flow
   END_VAR
BEGIN
   // _DB_Header[0] : ▄▄▄▄▄▄▄▄▄▄▄▄▄▄▄▄▄▄▄▄▄▄▄▄▄▄▄▄▄▄▄▄▄ ＳＴＡＮＤＡＲＤ ▄▄
   // _DB_Header[2] : TITLE: INSTRUMENTATION — ANALOG INSTRUMENT READ, SCALE AND MONITOR
   // _DB_Header[4] : ▀▀▀▀▀▀▀▀▀▀▀▀▀▀▀▀▀▀▀▀▀▀▀▀▀▀▀▀▀▀▀▀▀▀▀▀▀▀▀▀▀▀▀▀
   // _DB_Header[5] : TYPE: DYNAMIC
   // _DB_Header[6] : ▄▄▄▄▄▄▄▄▄▄▄▄▄▄▄▄▄▄▄▄▄▄▄▄▄▄▄▄▄▄▄▄▄▄▄▄▄▄▄▄▄▄▄▄
   // _DB_Header[8] : This is the dynamic data block associated with the standard analog instrument read
   // _DB_Header[9] : block:
   // _DB_Header[10] : FC02001_StdInstAnalog
   // _DB_Header[12] : The dynamic data holds the current scaled value of the instrument, along with
   // _DB_Header[13] : any alarms, warnings or faults.
   // _DB_Header[15] : Each instrument is given the user data type:
   // _DB_Header[16] : UT22001_Dy_InstAnalog
   // _DB_Header[17] : This holds the full set of static configuration data for the instrument.
   // _DB_Header[19] : ━━━ ⬙⬙⬙⬙⬙⬙ ━━━
   // _DB_Header[21] : ▄▄▄▄▄▄▄▄▄▄▄▄▄▄▄▄▄▄▄▄▄▄▄▄▄▄▄▄▄▄▄▄▄▄▄▄▄▄▄▄▄▄▄▄
   // _DB_Header[22] : MODIFICATION HISTORY
   // _DB_Header[24] : This is a summary of the recent software modifications made to this block (most recent at top)
   // _DB_Header[26] : ―――――――――――――――――――――――――――――――――――――――――――
   // _DB_Header[27] : DATE REVISION MASTER BRANCH DEV
   // _DB_Header[28] : (nnn.amm) COMMIT TAG (Base ---> Merge) BRANCH Author
   // _DB_Header[29] : ———————————————————————————————————————————
   // _DB_Header[30] : 2024.05.16 003.000 D0017A-000.105 D0017 D0018 None M. Gledhill
   // _DB_Header[31] : FC02001 — RELEASED FOR USE
   // _DB_Header[32] : Merge back to master branch
   // _DB_Header[34] : 2024.05.11 002.801 D0017A-000.104 D0017 N/A D017A M. Gledhill
   // _DB_Header[35] : RAW_ANALOG changed to AI_RAW_SIGNAL
   // _DB_Header[36] : AI_RAW_DATA and AI_SCALE_DATA added and
   // _DB_Header[37] : copied to DYNAMIC_DATA (see db00801 SMDS)
   // _DB_Header[39] : 2022.04.16 002.000 D0011 D0010 D0011 None M. Gledhill
   // _DB_Header[40] : FC02001 — RELEASED FOR USE
   // _DB_Header[41] : Merge back to master branch
   // _DB_Header[43] : 2022.04.11 001.801 D0010A-000.801 D0010 N/A D010A M. Gledhill
   // _DB_Header[44] : Released for test (SCV)
   // _DB_Header[46] : 2022.04.08 001.102 D0010A-000.104 D0010 N/A D010A M. Gledhill
   // _DB_Header[47] : Comments updated
   // _DB_Header[49] : 2022.04.05 001.101 D0010A-000.103 D0010 N/A D010A M. Gledhill
   // _DB_Header[50] : Over and under range based on scaled signal
   // _DB_Header[51] : INFO_TYPE, cal_OR_Abs and cal_UR_Abs added
   // _DB_Header[52] : Comments updated and standardised
   // _DB_Header[53] : UDT variable names standardised
   // _DB_Header[55] : 2021.05.26 001.000 D0008 D0006 D0008 None M. Gledhill
   // _DB_Header[56] : FC02001 — RELEASED FOR USE
   // _DB_Header[57] : Merge back to master branch
   // _DB_Header[59] : 2021.05.24 000.801 D0006B-000.801 D0006 N/A D0006B M. Gledhill
   // _DB_Header[60] : FC02001 — Released for SMT
   // _DB_Header[62] : 2021.05.18 000.101 D0006B-000.101 D0006 N/A D0006B M. Gledhill
   // _DB_Header[63] : FC02001 Migration to VCS
   // _DB_Header[64] : ———————————————————————————————————————————
   // _DB_Header[65] : Where: nnn = Major revision
   // _DB_Header[66] : a = Type (1-7 Development, 8 Proving, 9 Qualification, 0 Release)
   // _DB_Header[67] : mm = Minor revision (must be 00 if a = 0)
   // _DB_Header[68] : Block properties version number should be set to nn.a (only one decimal place)
   // _DB_Header[70] : ██████████████ █ █ █ █ END █ █ █ █ ██████████████
   revInfo.REV_BLOCK := 'DB22001';
   revInfo.REV_NUMBER := '003.000';
   revInfo.REV_DATE := '2024-05-16';
   revInfo.REV_AUTHOR := 'M. Gledhill';
   FIC101.revInfo.REV_BLOCK := 'DB22001';
   FIC101.revInfo.REV_NUMBER := '000.801';
   FIC101.revInfo.REV_DATE := '2021-05-24';
   FIC101.revInfo.REV_AUTHOR := 'M. Gledhill';
END_DATA_BLOCK

DATA_BLOCK "DB11001_St_DevValveIsol"   // DB11001
TITLE = Static DB [Device Driver] — Isolating Valve
{ S7_Optimized_Access := 'TRUE' }
AUTHOR : M_Gledhill
FAMILY : DeviceDriver
NAME : St_StdDevValveIsol
VERSION : 1.0
// PRACTICAL SERIES AUTOMATION LIBRARY (PAL)   —   COPYRIGHT 2020 – M. GLEDHILL (MIT LICENCE)
//                   ———— ◆ ————
//  FOR DETAILED DOCUMENTATION — SELECT THE BLOCK IN THE PROJECT TREE AND PRESS SHIFT + F1
//  FULL ONLINE DOCUMENTATION IS AVAILABLE AT: https://practicalseries.com/2001-pal/index.html
// stored: AutoNumber false, DBAccessibleFromOPCUA true, IsOnlyStoredInLoadMemory false, IsRetainMemResEnabled false, IsWriteProtectedInAS false, MemoryReserve 100
   VAR
      _DB_Header { ExternalAccessible := 'False'; ExternalVisible := 'False'; ExternalWritable := 'False'} : Array[0..79] of Bool;   // STANDARD ANALOG INSTRUMENT READ
      __________0000_0 { ExternalAccessible := 'False'; ExternalVisible := 'False'; ExternalWritable := 'False'} : Bool := false;
      __________0000_1 { ExternalAccessible := 'False'; ExternalVisible := 'False'; ExternalWritable := 'False'} : Bool := false;   // ▀▀▀▀ DB CURRENT REVISION
      revInfo { ExternalWritable := 'False'; S7_SetPoint := 'True'} : "UT01000_St_SysRevision";
      __________0010_0 { ExternalAccessible := 'False'; ExternalVisible := 'False'; ExternalWritable := 'False'} : Bool := false;
      __________0010_1 { ExternalAccessible := 'False'; ExternalVisible := 'False'; ExternalWritable := 'False'} : Bool := false;   // ▀▀▀▀ ISOLATING VALVES
      V001 { ExternalWritable := 'False'} : "UT11001_St_DevValveIsol";   // Filter 1 backwash inlet
   END_VAR
BEGIN
   // _DB_Header[0] : ▀▀▀▀▀▀▀▀▀▀▀▀▀▀▀▀▀▀▀▀▀▀▀▀▀▀▀▀▀▀▀▀▀▀▀▀▀▀▀▀▀▀▀▀
   // _DB_Header[2] : TITLE: STANDARD — DEVICE DRIVER FOR AN ISOLATING VALVE
   // _DB_Header[4] : ▄▄▄▄▄▄▄▄▄▄▄▄▄▄▄▄▄▄▄▄▄▄▄▄▄▄▄▄▄▄▄▄▄▄▄▄▄▄▄▄▄▄▄▄
   // _DB_Header[5] : TYPE: STATIC
   // _DB_Header[6] : ▀▀▀▀▀▀▀▀▀▀▀▀▀▀▀▀▀▀▀▀▀▀▀▀▀▀▀▀▀▀▀▀▀▀▀▀▀▀▀▀▀▀▀▀
   // _DB_Header[8] : This is the static data block associated with the standard device driver for an isolating valve
   // _DB_Header[9] : block:
   // _DB_Header[10] : FC11001_StdDevValveIsol
   // _DB_Header[12] : The static data holds the configuration data for the device (normally open/closed,
   // _DB_Header[13] : limit switch and interlock configuration &c.)
   // _DB_Header[15] : Each instrument is given the user data type:
   // _DB_Header[16] : UT11001_St_DevValveIsol
   // _DB_Header[17] : This holds the full set of static configuration data for the device
   // _DB_Header[19] : ━━━ ⬙⬙⬙⬙⬙⬙ ━━━
   // _DB_Header[21] : ▄▄▄▄▄▄▄▄▄▄▄▄▄▄▄▄▄▄▄▄▄▄▄▄▄▄▄▄▄▄▄▄▄▄▄▄▄▄▄▄▄▄▄▄
   // _DB_Header[22] : MODIFICATION HISTORY
   // _DB_Header[24] : This is a summary of the recent software modifications made to this block (most recent at top)
   // _DB_Header[26] : ―――――――――――――――――――――――――――――――――――――――――――
   // _DB_Header[27] : DATE REVISION MASTER BRANCH DEV
   // _DB_Header[28] : (nnn.amm) COMMIT TAG (Base ---> Merge) BRANCH Author
   // _DB_Header[29] : ———————————————————————————————————————————
   // _DB_Header[30] : 2021.08.23 001.000 D0009 D0008 D0009 None M. Gledhill
   // _DB_Header[31] : FC11001 — RELEASED FOR USE
   // _DB_Header[32] : Merge back to master branch
   // _DB_Header[34] : 2021.08.17 000.801 D0008A-000.801 D0008 N/A D0008A M. Gledhill
   // _DB_Header[35] : FC11001 Released for SMT
   // _DB_Header[37] : 2021.08.10 000.103 D0008A-000.103 D0008 N/A D0008A M. Gledhill
   // _DB_Header[38] : FC11001 Incremental build
   // _DB_Header[40] : 2021.07.21 000.102 D0008A-000.102 D0008 N/A D0008A M. Gledhill
   // _DB_Header[41] : FC11001 Incremental build
   // _DB_Header[43] : 2021.07.08 000.101 D0008A-000.101 D0008 N/A D0008A M. Gledhill
   // _DB_Header[44] : FC11001 Block created
   // _DB_Header[45] : ———————————————————————————————————————————
   // _DB_Header[46] : Where: nnn = Major revision
   // _DB_Header[47] : a = Type (1-7 Development, 8 Proving, 9 Qualification, 0 Release)
   // _DB_Header[48] : mm = Minor revision (must be 00 if a = 0)
   // _DB_Header[49] : Block properties version number should be set to nn.a (only one decimal place)
   // _DB_Header[51] : ██████████████ █ █ █ █ END █ █ █ █ ██████████████
   revInfo.REV_BLOCK := 'DB11001';
   revInfo.REV_NUMBER := '001.000';
   revInfo.REV_DATE := '2021.08.23';
   revInfo.REV_AUTHOR := 'M. Gledhill';
   V001.CONFIG_FBK_OPEN_EN := true;
   V001.CONFIG_FBK_CLOSED_EN := true;
   V001.TIME_OPENING_MAX := 20.0;
   V001.TIME_CLOSING_MAX := 30.0;
   V001.TIME_DER_OPEN := 80.0;
   V001.TIME_DER_CLOSED := 90.0;
END_DATA_BLOCK

DATA_BLOCK "DB11011_St_DevValve3Way"   // DB11011
TITLE = Static DB [DEVICE DRIVER] — Three-Way Valve
{ S7_Optimized_Access := 'TRUE' }
AUTHOR : M_Gledhill
FAMILY : DeviceDriver
NAME : St_DevValve3Way
VERSION : 0.8
// PRACTICAL SERIES AUTOMATION LIBRARY (PAL)   —   COPYRIGHT 2020 – M. GLEDHILL (MIT LICENCE)
//                   ———— ◆ ————
// FULL ONLINE DOCUMENTATION IS AVAILABLE AT: https://practicalseries.com/2001-pal/index.html
// stored: AutoNumber false, DBAccessibleFromOPCUA true, IsOnlyStoredInLoadMemory false, IsRetainMemResEnabled false, IsWriteProtectedInAS false, MemoryReserve 100
   VAR
      _DB_Header { ExternalAccessible := 'False'; ExternalVisible := 'False'; ExternalWritable := 'False'} : Array[0..79] of Bool;   // Static DB [DEVICE DRIVER] — Three-way Valve
      __________0000_0 { ExternalAccessible := 'False'; ExternalVisible := 'False'; ExternalWritable := 'False'} : Bool := false;
      __________0000_1 { ExternalAccessible := 'False'; ExternalVisible := 'False'; ExternalWritable := 'False'} : Bool := false;   // ▀▀▀▀ DB CURRENT REVISION
      revInfo { ExternalWritable := 'False'; S7_SetPoint := 'True'} : "UT01000_St_SysRevision";   // Revision information
      __________0010_0 { ExternalAccessible := 'False'; ExternalVisible := 'False'; ExternalWritable := 'False'} : Bool := false;
      __________0010_1 { ExternalAccessible := 'False'; ExternalVisible := 'False'; ExternalWritable := 'False'} : Bool := false;   // ▀▀▀▀ THREE-WAY VALVES
      V001 { ExternalWritable := 'False'; S7_SetPoint := 'True'} : "UT11011_St_DevValve3Way";   // Filter 1 backwash divert
   END_VAR
BEGIN
   // _DB_Header[0] : ▄▄▄▄▄▄▄▄▄▄▄▄▄▄▄▄▄▄▄▄▄▄▄▄▄▄▄▄▄▄▄▄▄ ＳＴＡＮＤＡＲＤ ▄▄
   // _DB_Header[2] : TITLE: DEVICE DRIVER — THREE-WAY VALVE
   // _DB_Header[4] : ▀▀▀▀▀▀▀▀▀▀▀▀▀▀▀▀▀▀▀▀▀▀▀▀▀▀▀▀▀▀▀▀▀▀▀▀▀▀▀▀▀▀▀▀
   // _DB_Header[5] : TYPE: STATIC
   // _DB_Header[6] : ▄▄▄▄▄▄▄▄▄▄▄▄▄▄▄▄▄▄▄▄▄▄▄▄▄▄▄▄▄▄▄▄▄▄▄▄▄▄▄▄▄▄▄▄
   // _DB_Header[8] : This is the static data block associated with the standard device driver for a three-way valve
   // _DB_Header[9] : block:
   // _DB_Header[10] : FC11011_StdDevValve3Way
   // _DB_Header[12] : The static data holds the configuration data for the device ( limit switch and
   // _DB_Header[13] : interlock configuration &c.)
   // _DB_Header[15] : Each valve is given the user data type:
   // _DB_Header[16] : UT11011_St_DevValve3Way
   // _DB_Header[17] : This holds the full set of static configuration data for the device
   // _DB_Header[19] : ━━━ ⬙⬙⬙⬙⬙⬙ ━━━
   // _DB_Header[21] : ▄▄▄▄▄▄▄▄▄▄▄▄▄▄▄▄▄▄▄▄▄▄▄▄▄▄▄▄▄▄▄▄▄▄▄▄▄▄▄▄▄▄▄▄
   // _DB_Header[22] : MODIFICATION HISTORY
   // _DB_Header[24] : This is a summary of the recent software modifications made to this block (most recent at top)
   // _DB_Header[26] : ―――――――――――――――――――――――――――――――――――――――――――
   // _DB_Header[27] : DATE REVISION MASTER BRANCH DEV
   // _DB_Header[28] : (nnn.amm) COMMIT TAG (Base ---> Merge) BRANCH Author
   // _DB_Header[29] : ———————————————————————————————————————————
   // _DB_Header[30] : 2022.06.07 000.801 D0014A-000.801 D0014 N/A D0014A M. Gledhill
   // _DB_Header[31] : Released for test (SMTS)
   // _DB_Header[33] : 2022.06.01 000.101 D0014A-000.101 D0014 N/A D0014A M. Gledhill
   // _DB_Header[34] : FC11011 Block created
   // _DB_Header[35] : ———————————————————————————————————————————
   // _DB_Header[36] : Where: nnn = Major revision
   // _DB_Header[37] : a = Type (1-7 Development, 8 Proving, 9 Qualification, 0 Release)
   // _DB_Header[38] : mm = Minor revision (must be 00 if a = 0)
   // _DB_Header[39] : Block properties version number should be set to nn.a (only one decimal place)
   // _DB_Header[41] : ██████████████ █ █ █ █ END █ █ █ █ ██████████████
   revInfo.REV_BLOCK := 'DB11011';
   revInfo.REV_NUMBER := '000.801';
   revInfo.REV_DATE := '2022.06.07';
   revInfo.REV_AUTHOR := 'M. Gledhill';
   V001.CONFIG_FBK_ENG_EN := true;
   V001.CONFIG_FBK_DENG_EN := true;
   V001.INFO_TAG := 'V001';
   V001.TIME_ENG_MAX := 20.0;
   V001.TIME_DENG_MAX := 30.0;
   V001.TIME_DER_ENG := 80.0;
   V001.TIME_DER_DENG := 90.0;
END_DATA_BLOCK

DATA_BLOCK "DB11101_St_DevValveBi"   // DB11101
TITLE = Static DB [DEVICE DRIVER] — Bistable Valve
{ S7_Optimized_Access := 'TRUE' }
AUTHOR : M_Gledhill
FAMILY : DeviceDriver
NAME : St_DevValveBi
VERSION : 0.8
// PRACTICAL SERIES AUTOMATION LIBRARY (PAL)   —   COPYRIGHT 2020 – M. GLEDHILL (MIT LICENCE)
//                   ———— ◆ ————
// FULL ONLINE DOCUMENTATION IS AVAILABLE AT: https://practicalseries.com/2001-pal/index.html
// stored: AutoNumber false, DBAccessibleFromOPCUA true, IsOnlyStoredInLoadMemory false, IsRetainMemResEnabled false, IsWriteProtectedInAS false, MemoryReserve 100
   VAR
      _DB_Header { ExternalAccessible := 'False'; ExternalVisible := 'False'; ExternalWritable := 'False'} : Array[0..79] of Bool;   // Static DB [DEVICE DRIVER] — Bistable Valve
      __________0000_0 { ExternalAccessible := 'False'; ExternalVisible := 'False'; ExternalWritable := 'False'} : Bool := false;
      __________0000_1 { ExternalAccessible := 'False'; ExternalVisible := 'False'; ExternalWritable := 'False'} : Bool := false;   // ▀▀▀▀ DB CURRENT REVISION
      revInfo { ExternalWritable := 'False'; S7_SetPoint := 'True'} : "UT01000_St_SysRevision";   // Revision information
      __________0010_0 { ExternalAccessible := 'False'; ExternalVisible := 'False'; ExternalWritable := 'False'} : Bool := false;
      __________0010_1 { ExternalAccessible := 'False'; ExternalVisible := 'False'; ExternalWritable := 'False'} : Bool := false;   // ▀▀▀▀ ISOLATING VALVES
      V001 { ExternalWritable := 'False'} : "UT11101_St_DevValveBi";   // Filter 1 backwash inlet
   END_VAR
BEGIN
   // _DB_Header[0] : ▄▄▄▄▄▄▄▄▄▄▄▄▄▄▄▄▄▄▄▄▄▄▄▄▄▄▄▄▄▄▄▄▄ ＳＴＡＮＤＡＲＤ ▄▄
   // _DB_Header[2] : TITLE: DEVICE DRIVER — BISTABLE VALVE
   // _DB_Header[4] : ▀▀▀▀▀▀▀▀▀▀▀▀▀▀▀▀▀▀▀▀▀▀▀▀▀▀▀▀▀▀▀▀▀▀▀▀▀▀▀▀▀▀▀▀
   // _DB_Header[5] : TYPE: STATIC
   // _DB_Header[6] : ▄▄▄▄▄▄▄▄▄▄▄▄▄▄▄▄▄▄▄▄▄▄▄▄▄▄▄▄▄▄▄▄▄▄▄▄▄▄▄▄▄▄▄▄
   // _DB_Header[8] : This is the static data block associated with the standard device driver for a bistable valve
   // _DB_Header[9] : block:
   // _DB_Header[10] : FC11101_StdDevValveBi
   // _DB_Header[12] : The static data holds the configuration data for the device (timer presets,
   // _DB_Header[13] : limit switch and interlock configuration &c.)
   // _DB_Header[15] : Each valve is given the user data type:
   // _DB_Header[16] : UT11101_St_DevValveBi
   // _DB_Header[17] : This holds the full set of static configuration data for the device
   // _DB_Header[19] : ━━━ ⬙⬙⬙⬙⬙⬙ ━━━
   // _DB_Header[21] : ▄▄▄▄▄▄▄▄▄▄▄▄▄▄▄▄▄▄▄▄▄▄▄▄▄▄▄▄▄▄▄▄▄▄▄▄▄▄▄▄▄▄▄▄
   // _DB_Header[22] : MODIFICATION HISTORY
   // _DB_Header[24] : This is a summary of the recent software modifications made to this block (most recent at top)
   // _DB_Header[26] : ―――――――――――――――――――――――――――――――――――――――――――
   // _DB_Header[27] : DATE REVISION MASTER BRANCH DEV
   // _DB_Header[28] : (nnn.amm) COMMIT TAG (Base ---> Merge) BRANCH Author
   // _DB_Header[29] : ———————————————————————————————————————————
   // _DB_Header[30] : 2023.02.01 000.801 D0015A-000.801 D0015 N/A D0015A M. Gledhill
   // _DB_Header[31] : FC11101 — Released for test (SMTS)
   // _DB_Header[33] : 2023.01.28 000.102 D0015A-000.102 D0015 N/A D0015A M. Gledhill
   // _DB_Header[34] : FC11101 — Incremental build
   // _DB_Header[36] : 2022.08.15 000.101 D0015A-000.101 D0008 N/A D0015A M. Gledhill
   // _DB_Header[37] : FC11101 Block created
   // _DB_Header[38] : ———————————————————————————————————————————
   // _DB_Header[39] : Where: nnn = Major revision
   // _DB_Header[40] : a = Type (1-7 Development, 8 Proving, 9 Qualification, 0 Release)
   // _DB_Header[41] : mm = Minor revision (must be 00 if a = 0)
   // _DB_Header[42] : Block properties version number should be set to nn.a (only one decimal place)
   // _DB_Header[44] : ██████████████ █ █ █ █ END █ █ █ █ ██████████████
   revInfo.REV_BLOCK := 'DB11101';
   revInfo.REV_NUMBER := '000.801';
   revInfo.REV_DATE := '2023.02.01';
   revInfo.REV_AUTHOR := 'M. Gledhill';
END_DATA_BLOCK

DATA_BLOCK "DB31001_Dy_DevValveIsol"   // DB31001
TITLE = Dynamic DB [DEVICE DRIVER] — Isolating Valve
{ S7_Optimized_Access := 'TRUE' }
AUTHOR : M_Gledhill
FAMILY : DeviceDriver
NAME : Dy_DevValveIsol
VERSION : 1.8
// PRACTICAL SERIES AUTOMATION LIBRARY (PAL)   —   COPYRIGHT 2020 – M. GLEDHILL (MIT LICENCE)
//                   ———— ◆ ————
// FULL ONLINE DOCUMENTATION IS AVAILABLE AT: https://practicalseries.com/2001-pal/index.html
// stored: AutoNumber false, DBAccessibleFromOPCUA true, IsOnlyStoredInLoadMemory false, IsRetainMemResEnabled false, IsWriteProtectedInAS false, MemoryReserve 100
   VAR
      _DB_Header { ExternalAccessible := 'False'; ExternalVisible := 'False'; ExternalWritable := 'False'} : Array[0..79] of Bool;   // Dynamic DB [DEVICE DRIVER] — Isolating Valve
      __________0000_0 { ExternalAccessible := 'False'; ExternalVisible := 'False'; ExternalWritable := 'False'} : Bool := false;
      __________0000_1 { ExternalAccessible := 'False'; ExternalVisible := 'False'; ExternalWritable := 'False'} : Bool := false;   // ▀▀▀▀ DB CURRENT REVISION
      revInfo { ExternalWritable := 'False'; S7_SetPoint := 'True'} : "UT01000_St_SysRevision";   // Revision information
      __________0010_0 { ExternalAccessible := 'False'; ExternalVisible := 'False'; ExternalWritable := 'False'} : Bool := false;
      __________0010_1 { ExternalAccessible := 'False'; ExternalVisible := 'False'; ExternalWritable := 'False'} : Bool := false;   // ▀▀▀▀ ISOLATING VALVES
      V001 { ExternalWritable := 'False'} : "UT31001_Dy_DevValveIsol";   // Filter 1 backwash inlet
   END_VAR
BEGIN
   // _DB_Header[0] : ▄▄▄▄▄▄▄▄▄▄▄▄▄▄▄▄▄▄▄▄▄▄▄▄▄▄▄▄▄▄▄▄▄ ＳＴＡＮＤＡＲＤ ▄▄
   // _DB_Header[2] : TITLE: DEVICE DRIVER — ISOLATING VALVE
   // _DB_Header[4] : ▀▀▀▀▀▀▀▀▀▀▀▀▀▀▀▀▀▀▀▀▀▀▀▀▀▀▀▀▀▀▀▀▀▀▀▀▀▀▀▀▀▀▀▀
   // _DB_Header[5] : TYPE: DYNAMIC
   // _DB_Header[6] : ▄▄▄▄▄▄▄▄▄▄▄▄▄▄▄▄▄▄▄▄▄▄▄▄▄▄▄▄▄▄▄▄▄▄▄▄▄▄▄▄▄▄▄▄
   // _DB_Header[8] : This is the dynamic data block associated with the standard device driver for an isolating valve
   // _DB_Header[9] : block:
   // _DB_Header[10] : FC11001_StdDevValveIsol
   // _DB_Header[12] : The dynamic data holds the live data for the device (its mode, status and messages
   // _DB_Header[13] : and any other dynamic information required by the module)
   // _DB_Header[15] : Each valve is given the user data type:
   // _DB_Header[16] : UT31001_Dy_DevValveIsol
   // _DB_Header[17] : This holds the full set of dynamic data for the device
   // _DB_Header[19] : ━━━ ⬙⬙⬙⬙⬙⬙ ━━━
   // _DB_Header[21] : ▄▄▄▄▄▄▄▄▄▄▄▄▄▄▄▄▄▄▄▄▄▄▄▄▄▄▄▄▄▄▄▄▄▄▄▄▄▄▄▄▄▄▄▄
   // _DB_Header[22] : MODIFICATION HISTORY
   // _DB_Header[24] : This is a summary of the recent software modifications made to this block (most recent at top)
   // _DB_Header[26] : ―――――――――――――――――――――――――――――――――――――――――――
   // _DB_Header[27] : DATE REVISION MASTER BRANCH DEV
   // _DB_Header[28] : (nnn.amm) COMMIT TAG (Base ---> Merge) BRANCH Author
   // _DB_Header[29] : ———————————————————————————————————————————
   // _DB_Header[30] : 2022.04.11 001.801 D0010A-000.801 D0010 N/A D010A M. Gledhill
   // _DB_Header[31] : Released for test (SCV)
   // _DB_Header[33] : 2022.04.06 001.101 D0010A-000.104 D0010 N/A D010A M. Gledhill
   // _DB_Header[34] : Comments updated and standardised
   // _DB_Header[36] : 2021.08.23 001.000 D0009 D0008 D0009 None M. Gledhill
   // _DB_Header[37] : FC11001 — RELEASED FOR USE
   // _DB_Header[38] : Merge back to master branch
   // _DB_Header[40] : 2021.08.17 000.801 D0008A-000.801 D0008 N/A D0008A M. Gledhill
   // _DB_Header[41] : FC11001 Released for SMT
   // _DB_Header[43] : 2021.08.10 000.103 D0008A-000.103 D0008 N/A D0008A M. Gledhill
   // _DB_Header[44] : FC11001 Incremental build
   // _DB_Header[46] : 2021.07.21 000.102 D0008A-000.102 D0008 N/A D0008A M. Gledhill
   // _DB_Header[47] : FC11001 Incremental build
   // _DB_Header[49] : 2021.07.08 000.101 D0008A-000.101 D0008 N/A D0008A M. Gledhill
   // _DB_Header[50] : FC11001 Block created
   // _DB_Header[51] : ———————————————————————————————————————————
   // _DB_Header[52] : Where: nnn = Major revision
   // _DB_Header[53] : a = Type (1-7 Development, 8 Proving, 9 Qualification, 0 Release)
   // _DB_Header[54] : mm = Minor revision (must be 00 if a = 0)
   // _DB_Header[55] : Block properties version number should be set to nn.a (only one decimal place)
   // _DB_Header[57] : ██████████████ █ █ █ █ END █ █ █ █ ██████████████
   revInfo.REV_BLOCK := 'DB31001';
   revInfo.REV_NUMBER := '001.801';
   revInfo.REV_DATE := '2022.04.11';
   revInfo.REV_AUTHOR := 'M. Gledhill';
END_DATA_BLOCK

DATA_BLOCK "DB31011_Dy_DevValve3Way"   // DB31011
TITLE = Dynamic DB [DEVICE DRIVER] — Three-Way Valve
{ S7_Optimized_Access := 'TRUE' }
AUTHOR : M_Gledhill
FAMILY : DeviceDriver
NAME : Dy_DevValve3Way
VERSION : 1.0
// PRACTICAL SERIES AUTOMATION LIBRARY (PAL)   —   COPYRIGHT 2020 – M. GLEDHILL (MIT LICENCE)
//                   ———— ◆ ————
// FULL ONLINE DOCUMENTATION IS AVAILABLE AT: https://practicalseries.com/2001-pal/index.html
// stored: AutoNumber false, DBAccessibleFromOPCUA true, IsOnlyStoredInLoadMemory false, IsRetainMemResEnabled false, IsWriteProtectedInAS false, MemoryReserve 100
   VAR
      _DB_Header { ExternalAccessible := 'False'; ExternalVisible := 'False'; ExternalWritable := 'False'} : Array[0..79] of Bool;   // Dynamic DB [DEVICE DRIVER] — Three-way Valve
      __________0000_0 { ExternalAccessible := 'False'; ExternalVisible := 'False'; ExternalWritable := 'False'} : Bool := false;
      __________0000_1 { ExternalAccessible := 'False'; ExternalVisible := 'False'; ExternalWritable := 'False'} : Bool := false;   // ▀▀▀▀ DB CURRENT REVISION
      revInfo { ExternalWritable := 'False'; S7_SetPoint := 'True'} : "UT01000_St_SysRevision";   // Revision information
      __________0010_0 { ExternalAccessible := 'False'; ExternalVisible := 'False'; ExternalWritable := 'False'} : Bool := false;
      __________0010_1 { ExternalAccessible := 'False'; ExternalVisible := 'False'; ExternalWritable := 'False'} : Bool := false;   // ▀▀▀▀ THREE-WAY VALVES
      V001 { ExternalWritable := 'False'} : "UT31011_Dy_DevValve3Way";   // Filter 1 backwash divert
   END_VAR
BEGIN
   // _DB_Header[0] : ▄▄▄▄▄▄▄▄▄▄▄▄▄▄▄▄▄▄▄▄▄▄▄▄▄▄▄▄▄▄▄▄▄ ＳＴＡＮＤＡＲＤ ▄▄
   // _DB_Header[2] : TITLE: DEVICE DRIVER — THREE-WAY VALVE
   // _DB_Header[4] : ▀▀▀▀▀▀▀▀▀▀▀▀▀▀▀▀▀▀▀▀▀▀▀▀▀▀▀▀▀▀▀▀▀▀▀▀▀▀▀▀▀▀▀▀
   // _DB_Header[5] : TYPE: DYNAMIC
   // _DB_Header[6] : ▄▄▄▄▄▄▄▄▄▄▄▄▄▄▄▄▄▄▄▄▄▄▄▄▄▄▄▄▄▄▄▄▄▄▄▄▄▄▄▄▄▄▄▄
   // _DB_Header[8] : This is the dynamic data block associated with the standard device driver for a three-way valve
   // _DB_Header[9] : block:
   // _DB_Header[10] : FC11011_StdDevValve3Way
   // _DB_Header[12] : The dynamic data holds the live data for the device (its mode, status and messages
   // _DB_Header[13] : and any other dynamic information required by the module)
   // _DB_Header[15] : Each valve is given the user data type:
   // _DB_Header[16] : UT31011_Dy_DevValve3Way
   // _DB_Header[17] : This holds the full set of dynamic data for the device
   // _DB_Header[19] : ━━━ ⬙⬙⬙⬙⬙⬙ ━━━
   // _DB_Header[21] : ▄▄▄▄▄▄▄▄▄▄▄▄▄▄▄▄▄▄▄▄▄▄▄▄▄▄▄▄▄▄▄▄▄▄▄▄▄▄▄▄▄▄▄▄
   // _DB_Header[22] : MODIFICATION HISTORY
   // _DB_Header[24] : This is a summary of the recent software modifications made to this block (most recent at top)
   // _DB_Header[26] : ―――――――――――――――――――――――――――――――――――――――――――
   // _DB_Header[27] : DATE REVISION MASTER BRANCH DEV
   // _DB_Header[28] : (nnn.amm) COMMIT TAG (Base ---> Merge) BRANCH Author
   // _DB_Header[29] : ———————————————————————————————————————————
   // _DB_Header[30] : 2022.06.11 001.000 D0015 D0014 D0015 None M. Gledhill
   // _DB_Header[31] : FC11011 — RELEASED FOR USE
   // _DB_Header[32] : Merge back to master branch
   // _DB_Header[34] : 2022.06.07 000.801 D0014A-000.801 D0014 N/A D0014A M. Gledhill
   // _DB_Header[35] : Released for test (SMTS)
   // _DB_Header[37] : 2022.06.01 000.101 D0014A-000.101 D0014 N/A D0014A M. Gledhill
   // _DB_Header[38] : FC11011 Block created
   // _DB_Header[39] : ———————————————————————————————————————————
   // _DB_Header[40] : Where: nnn = Major revision
   // _DB_Header[41] : a = Type (1-7 Development, 8 Proving, 9 Qualification, 0 Release)
   // _DB_Header[42] : mm = Minor revision (must be 00 if a = 0)
   // _DB_Header[43] : Block properties version number should be set to nn.a (only one decimal place)
   // _DB_Header[45] : ██████████████ █ █ █ █ END █ █ █ █ ██████████████
   revInfo.REV_BLOCK := 'DB31011';
   revInfo.REV_NUMBER := '001.000';
   revInfo.REV_DATE := '2022.06.11';
   revInfo.REV_AUTHOR := 'M. Gledhill';
END_DATA_BLOCK

DATA_BLOCK "DB31101_Dy_DevValveBi"   // DB31101
TITLE = Dynamic DB [DEVICE DRIVER] — Bistable Valve
{ S7_Optimized_Access := 'TRUE' }
AUTHOR : M_Gledhill
FAMILY : DeviceDriver
NAME : Dy_DevValveBi
VERSION : 1.0
// PRACTICAL SERIES AUTOMATION LIBRARY (PAL)   —   COPYRIGHT 2020 – M. GLEDHILL (MIT LICENCE)
//                   ———— ◆ ————
// FULL ONLINE DOCUMENTATION IS AVAILABLE AT: https://practicalseries.com/2001-pal/index.html
// stored: AutoNumber false, DBAccessibleFromOPCUA true, IsOnlyStoredInLoadMemory false, IsRetainMemResEnabled false, IsWriteProtectedInAS false, MemoryReserve 100
   VAR
      _DB_Header { ExternalAccessible := 'False'; ExternalVisible := 'False'; ExternalWritable := 'False'} : Array[0..79] of Bool;   // Dynamic DB [DEVICE DRIVER] — Bistable Valve
      __________0000_0 { ExternalAccessible := 'False'; ExternalVisible := 'False'; ExternalWritable := 'False'} : Bool := false;
      __________0000_1 { ExternalAccessible := 'False'; ExternalVisible := 'False'; ExternalWritable := 'False'} : Bool := false;   // ▀▀▀▀ DB CURRENT REVISION
      revInfo { ExternalWritable := 'False'; S7_SetPoint := 'True'} : "UT01000_St_SysRevision";   // Revision information
      __________0010_0 { ExternalAccessible := 'False'; ExternalVisible := 'False'; ExternalWritable := 'False'} : Bool := false;
      __________0010_1 { ExternalAccessible := 'False'; ExternalVisible := 'False'; ExternalWritable := 'False'} : Bool := false;   // ▀▀▀▀ ISOLATING VALVES
      V001 { ExternalWritable := 'False'} : "UT31101_Dy_DevValveBi";   // Filter 1 backwash inlet
   END_VAR
BEGIN
   // _DB_Header[0] : ▄▄▄▄▄▄▄▄▄▄▄▄▄▄▄▄▄▄▄▄▄▄▄▄▄▄▄▄▄▄▄▄▄ ＳＴＡＮＤＡＲＤ ▄▄
   // _DB_Header[2] : TITLE: DEVICE DRIVER — BISTABLE VALVE
   // _DB_Header[4] : ▀▀▀▀▀▀▀▀▀▀▀▀▀▀▀▀▀▀▀▀▀▀▀▀▀▀▀▀▀▀▀▀▀▀▀▀▀▀▀▀▀▀▀▀
   // _DB_Header[5] : TYPE: DYNAMIC
   // _DB_Header[6] : ▄▄▄▄▄▄▄▄▄▄▄▄▄▄▄▄▄▄▄▄▄▄▄▄▄▄▄▄▄▄▄▄▄▄▄▄▄▄▄▄▄▄▄▄
   // _DB_Header[8] : This is the dynamic data block associated with the standard device driver for an isolating valve
   // _DB_Header[9] : block:
   // _DB_Header[10] : FC11101_StdDevValveBi
   // _DB_Header[12] : The dynamic data holds the live data for the device (its mode, status and messages
   // _DB_Header[13] : and any other dynamic information required by the module)
   // _DB_Header[15] : Each valve is given the user data type:
   // _DB_Header[16] : UT31101_Dy_DevValveBi
   // _DB_Header[17] : This holds the full set of dynamic data for the device
   // _DB_Header[19] : ━━━ ⬙⬙⬙⬙⬙⬙ ━━━
   // _DB_Header[21] : ▄▄▄▄▄▄▄▄▄▄▄▄▄▄▄▄▄▄▄▄▄▄▄▄▄▄▄▄▄▄▄▄▄▄▄▄▄▄▄▄▄▄▄▄
   // _DB_Header[22] : MODIFICATION HISTORY
   // _DB_Header[24] : This is a summary of the recent software modifications made to this block (most recent at top)
   // _DB_Header[26] : ―――――――――――――――――――――――――――――――――――――――――――
   // _DB_Header[27] : DATE REVISION MASTER BRANCH DEV
   // _DB_Header[28] : (nnn.amm) COMMIT TAG (Base ---> Merge) BRANCH Author
   // _DB_Header[29] : ———————————————————————————————————————————
   // _DB_Header[30] : 2023.02.02 001.000 D0016 D0015 D0016 None M. Gledhill
   // _DB_Header[31] : FC11101 — RELEASED FOR USE
   // _DB_Header[32] : Merge back to master branch
   // _DB_Header[34] : 2023.02.01 000.801 D0015A-000.801 D0015 N/A D0015A M. Gledhill
   // _DB_Header[35] : FC11101 — Released for test (SMTS)
   // _DB_Header[37] : 2023.01.28 000.102 D0015A-000.102 D0015 N/A D0015A M. Gledhill
   // _DB_Header[38] : FC11101 — Incremental build
   // _DB_Header[40] : 2022.08.15 000.101 D0015A-000.101 D0008 N/A D0015A M. Gledhill
   // _DB_Header[41] : FC11101 Block created
   // _DB_Header[42] : ———————————————————————————————————————————
   // _DB_Header[43] : Where: nnn = Major revision
   // _DB_Header[44] : a = Type (1-7 Development, 8 Proving, 9 Qualification, 0 Release)
   // _DB_Header[45] : mm = Minor revision (must be 00 if a = 0)
   // _DB_Header[46] : Block properties version number should be set to nn.a (only one decimal place)
   // _DB_Header[48] : ██████████████ █ █ █ █ END █ █ █ █ ██████████████
   revInfo.REV_BLOCK := 'DB31101';
   revInfo.REV_NUMBER := '001.000';
   revInfo.REV_DATE := '2023.02.02';
   revInfo.REV_AUTHOR := 'M. Gledhill';
END_DATA_BLOCK

DATA_BLOCK "DB39511_Dy_DebugInst1Order"   // DB39511
TITLE = Dynamic DB [DEBUG] — First Order Response Simulation
{ S7_Optimized_Access := 'TRUE' }
AUTHOR : M_Gledhill
FAMILY : Debug
NAME : Dy_DebugInst1Order
VERSION : 0.1
// PRACTICAL SERIES AUTOMATION LIBRARY (PAL)   —   COPYRIGHT 2020 – M. GLEDHILL (MIT LICENCE)
//                   ———— ◆ ————
// FULL ONLINE DOCUMENTATION IS AVAILABLE AT: https://practicalseries.com/2001-pal/index.html
// stored: AutoNumber false, DBAccessibleFromOPCUA true, IsOnlyStoredInLoadMemory false, IsRetainMemResEnabled false, IsWriteProtectedInAS false, MemoryReserve 100
   VAR
      _DB_Header { ExternalAccessible := 'False'; ExternalVisible := 'False'; ExternalWritable := 'False'} : Array[0..79] of Bool;   // Dynamic DB [DEBUG] — First Order Response Simulation
      __________0000_0 { ExternalAccessible := 'False'; ExternalVisible := 'False'; ExternalWritable := 'False'} : Bool := false;
      __________0000_1 { ExternalAccessible := 'False'; ExternalVisible := 'False'; ExternalWritable := 'False'} : Bool := false;   // ▀▀▀▀ DB CURRENT REVISION
      revInfo { ExternalWritable := 'False'; S7_SetPoint := 'True'} : "UT01000_St_SysRevision";   // Revision information
      __________0010_0 { ExternalAccessible := 'False'; ExternalVisible := 'False'; ExternalWritable := 'False'} : Bool := false;
      __________0010_1 { ExternalAccessible := 'False'; ExternalVisible := 'False'; ExternalWritable := 'False'} : Bool := false;   // ▀▀▀▀ 2ND ORDER SIMULATION
      SIM001 { ExternalWritable := 'False'} : "UT39511_Dy_DebugInst1Order";   // Simulation 001
   END_VAR
BEGIN
   // _DB_Header[0] : ▄▄▄▄▄▄▄▄▄▄▄▄▄▄▄▄▄▄▄▄▄▄▄▄▄▄▄▄▄▄▄▄▄ ＳＴＡＮＤＡＲＤ ▄▄
   // _DB_Header[2] : TITLE: DEBUG — FIRST ORDER RESPONSE SIMULATION
   // _DB_Header[4] : ▀▀▀▀▀▀▀▀▀▀▀▀▀▀▀▀▀▀▀▀▀▀▀▀▀▀▀▀▀▀▀▀▀▀▀▀▀▀▀▀▀▀▀▀
   // _DB_Header[5] : TYPE: DYNAMIC
   // _DB_Header[6] : ▄▄▄▄▄▄▄▄▄▄▄▄▄▄▄▄▄▄▄▄▄▄▄▄▄▄▄▄▄▄▄▄▄▄▄▄▄▄▄▄▄▄▄▄
   // _DB_Header[8] : This is the dynamic data block associated with the standard DEBUG
   // _DB_Header[9] : First Order Response Simulation function block:
   // _DB_Header[10] : FC19511_StdDebugInst1Order
   // _DB_Header[12] : The dynamic data holds live data such as calculation variables, simulation elapsed time,
   // _DB_Header[13] : status signals and any other information required by the module
   // _DB_Header[15] : Each simulation is given the user data type:
   // _DB_Header[16] : UT39511_Dy_DebugInst1Order
   // _DB_Header[17] : This holds the full set of dynamic data for the simulation
   // _DB_Header[19] : ━━━ ⬙⬙⬙⬙⬙⬙ ━━━
   // _DB_Header[21] : ▄▄▄▄▄▄▄▄▄▄▄▄▄▄▄▄▄▄▄▄▄▄▄▄▄▄▄▄▄▄▄▄▄▄▄▄▄▄▄▄▄▄▄▄
   // _DB_Header[22] : MODIFICATION HISTORY
   // _DB_Header[24] : This is a summary of the recent software modifications made to this block (most recent at top)
   // _DB_Header[26] : ―――――――――――――――――――――――――――――――――――――――――――
   // _DB_Header[27] : DATE REVISION MASTER BRANCH DEV
   // _DB_Header[28] : (nnn.amm) COMMIT TAG (Base ---> Merge) BRANCH Author
   // _DB_Header[29] : ———————————————————————————————————————————
   // _DB_Header[30] : 2023.02.26 000.101 D0016A-000.101 D0016 N/A D0016A M. Gledhill
   // _DB_Header[31] : FC19511 Block created
   // _DB_Header[32] : ———————————————————————————————————————————
   // _DB_Header[33] : Where: nnn = Major revision
   // _DB_Header[34] : a = Type (1-7 Development, 8 Proving, 9 Qualification, 0 Release)
   // _DB_Header[35] : mm = Minor revision (must be 00 if a = 0)
   // _DB_Header[36] : Block properties version number should be set to nn.a (only one decimal place)
   // _DB_Header[38] : ██████████████ █ █ █ █ END █ █ █ █ ██████████████
   revInfo.REV_BLOCK := 'DB39511';
   revInfo.REV_NUMBER := '000.101';
   revInfo.REV_DATE := '2023-02-26';
   revInfo.REV_AUTHOR := 'M. Gledhill';
END_DATA_BLOCK

DATA_BLOCK "DB39512_Dy_DebugInst2Order"   // DB39512
TITLE = Dynamic DB [DEBUG] — Second Order Response Simulation
{ S7_Optimized_Access := 'TRUE' }
AUTHOR : M_Gledhill
FAMILY : Debug
NAME : Dy_DebugInst2Order
VERSION : 1.1
// PRACTICAL SERIES AUTOMATION LIBRARY (PAL)   —   COPYRIGHT 2020 – M. GLEDHILL (MIT LICENCE)
//                   ———— ◆ ————
// FULL ONLINE DOCUMENTATION IS AVAILABLE AT: https://practicalseries.com/2001-pal/index.html
// stored: AutoNumber false, DBAccessibleFromOPCUA true, IsOnlyStoredInLoadMemory false, IsRetainMemResEnabled false, IsWriteProtectedInAS false, MemoryReserve 100
   VAR
      _DB_Header { ExternalAccessible := 'False'; ExternalVisible := 'False'; ExternalWritable := 'False'} : Array[0..79] of Bool;   // Dynamic DB [DEBUG] — Second Order Response Simulation
      __________0000_0 { ExternalAccessible := 'False'; ExternalVisible := 'False'; ExternalWritable := 'False'} : Bool := false;
      __________0000_1 { ExternalAccessible := 'False'; ExternalVisible := 'False'; ExternalWritable := 'False'} : Bool := false;   // ▀▀▀▀ DB CURRENT REVISION
      revInfo { ExternalWritable := 'False'; S7_SetPoint := 'True'} : "UT01000_St_SysRevision";   // Revision information
      __________0010_0 { ExternalAccessible := 'False'; ExternalVisible := 'False'; ExternalWritable := 'False'} : Bool := false;
      __________0010_1 { ExternalAccessible := 'False'; ExternalVisible := 'False'; ExternalWritable := 'False'} : Bool := false;   // ▀▀▀▀ 2ND ORDER SIMULATION
      SIM001 { ExternalWritable := 'False'} : "UT39512_Dy_DebugInst2Order";   // Simulation 001
   END_VAR
BEGIN
   // _DB_Header[0] : ▄▄▄▄▄▄▄▄▄▄▄▄▄▄▄▄▄▄▄▄▄▄▄▄▄▄▄▄▄▄▄▄▄ ＳＴＡＮＤＡＲＤ ▄▄
   // _DB_Header[2] : TITLE: DEBUG — SECOND ORDER RESPONSE SIMULATION
   // _DB_Header[4] : ▀▀▀▀▀▀▀▀▀▀▀▀▀▀▀▀▀▀▀▀▀▀▀▀▀▀▀▀▀▀▀▀▀▀▀▀▀▀▀▀▀▀▀▀
   // _DB_Header[5] : TYPE: DYNAMIC
   // _DB_Header[6] : ▄▄▄▄▄▄▄▄▄▄▄▄▄▄▄▄▄▄▄▄▄▄▄▄▄▄▄▄▄▄▄▄▄▄▄▄▄▄▄▄▄▄▄▄
   // _DB_Header[8] : This is the dynamic data block associated with the standard DEBUG
   // _DB_Header[9] : Second Order Response Simulation function block:
   // _DB_Header[10] : FC19512_StdDebugInst2Order
   // _DB_Header[12] : The dynamic data holds live data such as calculation variables, simulation elapsed time,
   // _DB_Header[13] : oscillation frequency, status signals and any other information required by the module
   // _DB_Header[15] : Each simulation is given the user data type:
   // _DB_Header[16] : UT39512_Dy_DebugInst2Order
   // _DB_Header[17] : This holds the full set of dynamic data for the simulation
   // _DB_Header[19] : ━━━ ⬙⬙⬙⬙⬙⬙ ━━━
   // _DB_Header[21] : ▄▄▄▄▄▄▄▄▄▄▄▄▄▄▄▄▄▄▄▄▄▄▄▄▄▄▄▄▄▄▄▄▄▄▄▄▄▄▄▄▄▄▄▄
   // _DB_Header[22] : MODIFICATION HISTORY
   // _DB_Header[24] : This is a summary of the recent software modifications made to this block (most recent at top)
   // _DB_Header[26] : ―――――――――――――――――――――――――――――――――――――――――――
   // _DB_Header[27] : DATE REVISION MASTER BRANCH DEV
   // _DB_Header[28] : (nnn.amm) COMMIT TAG (Base ---> Merge) BRANCH Author
   // _DB_Header[29] : ———————————————————————————————————————————
   // _DB_Header[30] : 2022.04.06 001.101 D0010A-000.104 D0010 N/A D010A M. Gledhill
   // _DB_Header[31] : Comments updated and standardised
   // _DB_Header[33] : 2022.03.04 001.000 D0010 D0009 D0010 None M. Gledhill
   // _DB_Header[34] : FC19512 — RELEASED FOR USE
   // _DB_Header[35] : Merge back to master branch
   // _DB_Header[37] : 2022.02.18 000.801 D0009A-000.801 D0009 N/A D0009A M. Gledhill
   // _DB_Header[38] : FC19512 Released for test
   // _DB_Header[40] : 2022.02.18 000.103 D0009A-000.103 D0009 N/A D0009A M. Gledhill
   // _DB_Header[41] : FC19512 Incremental build
   // _DB_Header[43] : 2022.02.02 000.102 D0009A-000.101 D0009 N/A D0009A M. Gledhill
   // _DB_Header[44] : FC19512 Incremental build
   // _DB_Header[45] : ———————————————————————————————————————————
   // _DB_Header[46] : Where: nnn = Major revision
   // _DB_Header[47] : a = Type (1-7 Development, 8 Proving, 9 Qualification, 0 Release)
   // _DB_Header[48] : mm = Minor revision (must be 00 if a = 0)
   // _DB_Header[49] : Block properties version number should be set to nn.a (only one decimal place)
   // _DB_Header[51] : ██████████████ █ █ █ █ END █ █ █ █ ██████████████
   revInfo.REV_BLOCK := 'DB39512';
   revInfo.REV_NUMBER := '001.101';
   revInfo.REV_DATE := '2022-04-06';
   revInfo.REV_AUTHOR := 'M. Gledhill';
END_DATA_BLOCK

DATA_BLOCK "DB18151_Dy_SubTimeEventRTC"   // DB18151
TITLE = Dynamic DB — Subroutine - Event Timer Using RTC
{ S7_Optimized_Access := 'TRUE' }
AUTHOR : M_Gledhill
FAMILY : Subroutine
NAME : Dy_SubTimeEventRTC
VERSION : 1.0
// PRACTICAL SERIES AUTOMATION LIBRARY (PAL)   —   COPYRIGHT 2020 – M. GLEDHILL (MIT LICENCE)
//                   ———— ◆ ————
//  FOR DETAILED DOCUMENTATION — SELECT THE BLOCK IN THE PROJECT TREE AND PRESS SHIFT + F1
//  FULL ONLINE DOCUMENTATION IS AVAILABLE AT: https://practicalseries.com/2001-pal/index.html
// stored: AutoNumber false, DBAccessibleFromOPCUA true, IsOnlyStoredInLoadMemory false, IsRetainMemResEnabled false, IsWriteProtectedInAS false, MemoryReserve 100
   VAR
      _DB_Header { ExternalAccessible := 'False'; ExternalVisible := 'False'; ExternalWritable := 'False'} : Array[0..79] of Bool;   // SUBROUTINE EVENT TIMER USING RTC
      __________0000_0 { ExternalWritable := 'False'} : Bool := false;
      __________0000_1 { ExternalWritable := 'False'} : Bool := false;   // ▀▀▀▀ DB CURRENT REVISION
      revInfo { ExternalWritable := 'False'} : "UT01000_St_SysRevision";
      __________0010_0 { ExternalAccessible := 'False'; ExternalVisible := 'False'; ExternalWritable := 'False'} : Bool := false;
      __________0010_1 { ExternalAccessible := 'False'; ExternalVisible := 'False'; ExternalWritable := 'False'} : Bool := false;   // ▀▀▀▀ SYSTEM EVENT TIMER
      FC18151_DayEvent { ExternalWritable := 'False'} : "UT18151_Dy_SubTimeEventRTC";   // Event timer — 1 Day
      FC18151_HourEvent { ExternalWritable := 'False'} : "UT18151_Dy_SubTimeEventRTC";   // Event timer — 1 Hour
      FC18151_MinEvent { ExternalWritable := 'False'} : "UT18151_Dy_SubTimeEventRTC";   // Event timer — 1 Minute
      FC18151_SecEvent { ExternalWritable := 'False'} : "UT18151_Dy_SubTimeEventRTC";   // Event timer — 1 Second
      FC18151_msEvent { ExternalWritable := 'False'} : "UT18151_Dy_SubTimeEventRTC";   // Event timer — 1 Millisecond
   END_VAR
BEGIN
   // _DB_Header[0] : ▀▀▀▀▀▀▀▀▀▀▀▀▀▀▀▀▀▀▀▀▀▀▀▀▀▀▀▀▀▀▀▀▀▀▀▀▀▀▀▀▀▀▀▀
   // _DB_Header[2] : TITLE: SUBROUTINE EVENT TIMER USING RTC
   // _DB_Header[4] : ▄▄▄▄▄▄▄▄▄▄▄▄▄▄▄▄▄▄▄▄▄▄▄▄▄▄▄▄▄▄▄▄▄▄▄▄▄▄▄▄▄▄▄▄
   // _DB_Header[5] : TYPE: DYNAMIC
   // _DB_Header[6] : ▀▀▀▀▀▀▀▀▀▀▀▀▀▀▀▀▀▀▀▀▀▀▀▀▀▀▀▀▀▀▀▀▀▀▀▀▀▀▀▀▀▀▀▀
   // _DB_Header[8] : This is the dynamic data block associated with the event timing subroutine block
   // _DB_Header[10] : FC18151_SubTimeEventRTC
   // _DB_Header[12] : The dynamic data holds the event start time, end time and duration
   // _DB_Header[14] : Each event is given the user data type:
   // _DB_Header[15] : UT18151_Dy_SubTimeEventRTC
   // _DB_Header[19] : ━━━ ⬙⬙⬙⬙⬙⬙ ━━━
   // _DB_Header[21] : ▄▄▄▄▄▄▄▄▄▄▄▄▄▄▄▄▄▄▄▄▄▄▄▄▄▄▄▄▄▄▄▄▄▄▄▄▄▄▄▄▄▄▄▄
   // _DB_Header[22] : MODIFICATION HISTORY
   // _DB_Header[24] : This is a summary of the recent software modifications made to this block (most recent at top)
   // _DB_Header[26] : ―――――――――――――――――――――――――――――――――――――――――――
   // _DB_Header[27] : DATE REVISION MASTER BRANCH DEV
   // _DB_Header[28] : (nnn.amm) COMMIT TAG (Base ---> Merge) BRANCH Author
   // _DB_Header[29] : ———————————————————————————————————————————
   // _DB_Header[30] : 2020.11.18 000.801 D0002A-000.801 D0002 N/A D0002A M. Gledhill
   // _DB_Header[31] : FC18151 Migration to VCS — Released for test
   // _DB_Header[32] : ———————————————————————————————————————————
   // _DB_Header[33] : Where: nnn = Major revision
   // _DB_Header[34] : a = Type (1-7 Development, 8 Proving, 9 Qualification, 0 Release)
   // _DB_Header[35] : mm = Minor revision (must be 00 if a = 0)
   // _DB_Header[36] : Block properties version number should be set to nn.a (only one decimal place)
   // _DB_Header[38] : ██████████████ █ █ █ █ END █ █ █ █ ██████████████
   revInfo.REV_BLOCK := 'DB18151';
   revInfo.REV_NUMBER := '001.000';
   revInfo.REV_DATE := '2021-02-18';
   revInfo.REV_AUTHOR := 'M. Gledhill';
END_DATA_BLOCK

DATA_BLOCK "DB38151_Dy_SubTimeEventRTC"   // DB38151
TITLE = Dynamic DB — Subroutine - Event Timer Using RTC
{ S7_Optimized_Access := 'TRUE' }
AUTHOR : M_Gledhill
FAMILY : Subroutine
NAME : Dy_SubTimeEventRTC
VERSION : 1.0
// PRACTICAL SERIES AUTOMATION LIBRARY (PAL)   —   COPYRIGHT 2020 – M. GLEDHILL (MIT LICENCE)
//                   ———— ◆ ————
//  FOR DETAILED DOCUMENTATION — SELECT THE BLOCK IN THE PROJECT TREE AND PRESS SHIFT + F1
//  FULL ONLINE DOCUMENTATION IS AVAILABLE AT: https://practicalseries.com/2001-pal/index.html
// stored: AutoNumber false, DBAccessibleFromOPCUA true, IsOnlyStoredInLoadMemory false, IsRetainMemResEnabled false, IsWriteProtectedInAS false, MemoryReserve 100
   VAR
      _DB_Header { ExternalAccessible := 'False'; ExternalVisible := 'False'; ExternalWritable := 'False'} : Array[0..79] of Bool;   // SUBROUTINE EVENT TIMER USING RTC
      __________0000_0 { ExternalWritable := 'False'} : Bool := false;
      __________0000_1 { ExternalWritable := 'False'} : Bool := false;   // ▀▀▀▀ DB CURRENT REVISION
      revInfo { ExternalWritable := 'False'} : "UT01000_St_SysRevision";
      __________0010_0 { ExternalAccessible := 'False'; ExternalVisible := 'False'; ExternalWritable := 'False'} : Bool := false;
      __________0010_1 { ExternalAccessible := 'False'; ExternalVisible := 'False'; ExternalWritable := 'False'} : Bool := false;   // ▀▀▀▀ SYSTEM EVENT TIMER
      FC18151_Event { ExternalWritable := 'False'} : "UT38151_Dy_SubTimeEventRTC";   // Event timer — 1 Day
      FC02001_AlmH_OnTime { ExternalWritable := 'False'; S7_SetPoint := 'True'} : "UT38151_Dy_SubTimeEventRTC";   // FC02001 Test — Alarm High On Time
      FC02001_AlmH_OffTime { ExternalWritable := 'False'; S7_SetPoint := 'True'} : "UT38151_Dy_SubTimeEventRTC";   // FC02001 Test — Alarm High Off Time
      FC02001_AlmL_OnTime { ExternalWritable := 'False'; S7_SetPoint := 'True'} : "UT38151_Dy_SubTimeEventRTC";   // FC02001 Test — Alarm Low On Time
      FC02001_AlmL_OffTime { ExternalWritable := 'False'; S7_SetPoint := 'True'} : "UT38151_Dy_SubTimeEventRTC";   // FC02001 Test — Alarm Low Off Time
      FC02001_WrnH_OnTime { ExternalWritable := 'False'; S7_SetPoint := 'True'} : "UT38151_Dy_SubTimeEventRTC";   // FC02001 Test — Warning High On Time
      FC02001_WrnH_OffTime { ExternalWritable := 'False'; S7_SetPoint := 'True'} : "UT38151_Dy_SubTimeEventRTC";   // FC02001 Test — Warning High Off Time
      FC02001_WrnL_OnTime { ExternalWritable := 'False'; S7_SetPoint := 'True'} : "UT38151_Dy_SubTimeEventRTC";   // FC02001 Test — Warning Low On Time
      FC02001_WrnL_OffTime { ExternalWritable := 'False'; S7_SetPoint := 'True'} : "UT38151_Dy_SubTimeEventRTC";   // FC02001 Test — Warning Low Off Time
   END_VAR
BEGIN
   // _DB_Header[0] : ▀▀▀▀▀▀▀▀▀▀▀▀▀▀▀▀▀▀▀▀▀▀▀▀▀▀▀▀▀▀▀▀▀▀▀▀▀▀▀▀▀▀▀▀
   // _DB_Header[2] : TITLE: SUBROUTINE EVENT TIMER USING RTC
   // _DB_Header[4] : ▄▄▄▄▄▄▄▄▄▄▄▄▄▄▄▄▄▄▄▄▄▄▄▄▄▄▄▄▄▄▄▄▄▄▄▄▄▄▄▄▄▄▄▄
   // _DB_Header[5] : TYPE: DYNAMIC
   // _DB_Header[6] : ▀▀▀▀▀▀▀▀▀▀▀▀▀▀▀▀▀▀▀▀▀▀▀▀▀▀▀▀▀▀▀▀▀▀▀▀▀▀▀▀▀▀▀▀
   // _DB_Header[8] : This is the dynamic data block associated with the event timing subroutine block
   // _DB_Header[10] : FC18151_SubTimeEventRTC
   // _DB_Header[12] : The dynamic data holds the event start time, end time and duration
   // _DB_Header[14] : Each event is given the user data type:
   // _DB_Header[15] : UT18151_Dy_SubTimeEventRTC
   // _DB_Header[19] : ━━━ ⬙⬙⬙⬙⬙⬙ ━━━
   // _DB_Header[21] : ▄▄▄▄▄▄▄▄▄▄▄▄▄▄▄▄▄▄▄▄▄▄▄▄▄▄▄▄▄▄▄▄▄▄▄▄▄▄▄▄▄▄▄▄
   // _DB_Header[22] : MODIFICATION HISTORY
   // _DB_Header[24] : This is a summary of the recent software modifications made to this block (most recent at top)
   // _DB_Header[26] : ―――――――――――――――――――――――――――――――――――――――――――
   // _DB_Header[27] : DATE REVISION MASTER BRANCH DEV
   // _DB_Header[28] : (nnn.amm) COMMIT TAG (Base ---> Merge) BRANCH Author
   // _DB_Header[29] : ———————————————————————————————————————————
   // _DB_Header[30] : 2021.02.19 001.000 D0003 D0002 D0003 None M. Gledhill
   // _DB_Header[31] : FC18151 — RELEASED FOR USE
   // _DB_Header[32] : Merge back to master branch
   // _DB_Header[34] : 2021.02.19 001.000 D0002A-001.000 D0002 N/A D0002A M. Gledhill
   // _DB_Header[35] : FC18151 — Post test RELEASED FOR USE
   // _DB_Header[37] : 2021.02.18 000.801 D0002A-000.801 D0002 N/A D0002A M. Gledhill
   // _DB_Header[38] : FC18151 Migration to VCS — Released for test
   // _DB_Header[39] : ———————————————————————————————————————————
   // _DB_Header[40] : Where: nnn = Major revision
   // _DB_Header[41] : a = Type (1-7 Development, 8 Proving, 9 Qualification, 0 Release)
   // _DB_Header[42] : mm = Minor revision (must be 00 if a = 0)
   // _DB_Header[43] : Block properties version number should be set to nn.a (only one decimal place)
   // _DB_Header[45] : ██████████████ █ █ █ █ END █ █ █ █ ██████████████
   revInfo.REV_BLOCK := 'DB38151';
   revInfo.REV_NUMBER := '001.000';
   revInfo.REV_DATE := '2021-02-19';
   revInfo.REV_AUTHOR := 'M. Gledhill';
END_DATA_BLOCK

ORGANIZATION_BLOCK "OB00001_IntINrmMainProgram"   // OB1, LAD, ProgramCycle
TITLE = Interrupt Module [NORMAL INTERRUPT] — Main Program Cyclic Execution
{ S7_Optimized_Access := 'TRUE' }
AUTHOR : M_Gledhill
FAMILY : Interrupt
NAME : IntINrmMainProgram
VERSION : 0.1
// PRACTICAL SERIES AUTOMATION LIBRARY (PAL)   —   COPYRIGHT 2020 – M. GLEDHILL (MIT LICENCE)
//                   ———— ◆ ————
// FULL ONLINE DOCUMENTATION IS AVAILABLE AT: https://practicalseries.com/2001-pal/index.html
// stored: AutoNumber true, IsIECCheckEnabled false, SetENOAutomatically false
   VAR_INPUT
      Initial_Call : Bool;   // Initial call of this OB
      Remanence : Bool;   // =True, if remanent data are available
   END_VAR
   VAR_TEMP
      revInfo : "UT01000_St_SysRevision";   // Revision information for this block
      licInfo : "UT01001_St_SysLicence";   // Licence information for this block
   END_VAR
BEGIN

REGION Network 1: Project description
   // ▄▄▄▄▄▄▄▄▄▄▄▄▄▄▄▄▄▄▄▄▄▄▄▄▄▄▄▄▄▄▄▄▄▄▄▄▄▄▄▄▄▄▄▄ 
   // 
   // 
   // TITLE:    PS2001 — PRACTICAL SERIES AUTOMATION LIBRARY
   // 
   // 
   // ▀▀▀▀▀▀▀▀▀▀▀▀▀▀▀▀▀▀▀▀▀▀▀▀▀▀▀▀▀▀▀▀▀▀▀▀▀▀▀▀▀▀▀▀ 
   // 
   // 
   // ――――――――――――――――――――――――――――――――――
   // COPYRIGHT:       © 2020 Michael Gledhill
   //           Part of the Practical Series of Publications
   //           Published in the United Kingdom
   //           mg@practicalseries.com
   //           https://practicalseries.com
   // ――――――――――――――――――――――――――――――――――
   // CUSTOMER:       Practical Series of Publications (PSP)
   // 
   // PROJECT:      Practical Series Automation Library (PAL)
   // 
   // PROJECT NO.:       PS2001
   // ――――――――――――――――――――――――――――――――――
   // CONTROLLER:       CPU 1515-2PN/DP
   // 
   // CONTROLLER NAME:    CON100
   // 
   // IP ADDRESS:      192.168.001.100
   // ――――――――――――――――――――――――――――――――――
   // TIA PROJECT NAME:    PS2001-PAL-D0018
   // STATUS:        DEVELOPMENT
   // ――――――――――――――――――――――――――――――――――
   // PROTECTION:     To minimise the risk of inadvertent modification to 
   //           tested modules, certain blocks will be released for 
   //           use with “protected access” (referred to a “write 
   //           protection” in Siemens terminology), this allows the 
   //           block to be used normally, but prevents the block 
   //           being accidentally modified. 
   // 
   //           This is in accordance with the risk assessment given 
   //           in the Validation Plant (VP), Appendix A [Ref. 002].
   // 
   //           ┌─────────────────────┐
   //           │ THE WRITE PROTECTION PASSWORD IS: PS2001 │
   //           └─────────────────────┘
   // 
   // 
   // ▄▄▄▄▄▄▄▄▄▄▄▄▄▄▄▄▄▄▄▄▄▄▄▄▄▄▄▄▄▄▄▄▄▄▄▄▄▄▄▄▄▄▄▄
   // PROJECT OVERVIEW
   // 
   // 
   // The PAL is a library of software modules and templates that have been developed for the 
   // Siemens Simatic S7-1500 range of controllers (and to a lesser extent the S7-1200 range).
   // 
   // The full library and all necessary documentation is available from the Practical Series website:
   // 
   //      https://practicalseries.com/2001-pal/index.html
   // 
   // 
   // The PAL is configured and deployed using the Siemens Simatic TIA Portal programming 
   // environment (version 16 or higher).
   // 
   // The PAL software structure is designed such that it is applicable to virtually all industrial 
   // applications that can generally controlled by a programmable logic controller.
   // 
   // The PAL software being developed as part of this Project, is considered to be suitable for use in 
   // the following types of industries (this is not an exhaustive list):
   // 
   //    •   Water and waste water treatment
   //    •   Pharmaceutical and batch production
   //    •   Brewing and fermentation
   //    •   Chemical manufacturing
   //    •   Oil and gas systems
   //    •   Food and beverage production
   // 
   // Such applications can generally be thought of as processes that operate with a response time
   // of more than 100 ms. I.e. the system would not be expected to respond to some stimuli faster
   // than 100 ms. In practice, a Controller may (and usually will) respond faster than this; however, 
   // a response time of 100 ms is considered to be an acceptable limit for PLC control.
   // 
   // At its most basic level, the PAL will be a library of software modules that control the fundamental 
   // aspects of an industrial plant; such modules would for example read the value of an instrument, 
   // operate a valve or drive, perform a calculation &c.
   // 
   // Such software modules are referred to as standard modules, these are fixed modules that 
   // perform a particular function and are identical across all software installations.
   // 
   // The PAL also contains application specific modules; these contain software that is applicable 
   // to the plant being controlled.
   // 
   // The Practical Series Automation Library is freely available under the MIT Open Source licence 
   // (see below). Those who find it useful may, if they wish, make a donation to support the library. 
   // 
   // Donations can be made here:
   // 
   //      https://practicalseries.com/2001-pal/11-web/81-00-pay.html
   // 
   // The PAL contains fully deployable software that has been developed by the author in his 
   // profession as a chartered electrical engineer. It is currently in use on various live plants 
   // throughout the UK and in some other parts of the world. 
   // 
   // This software is suitable for controlling and automating most industrial applications (typical 
   // process applications). It is easy to use and configure, but does have a degree of practical 
   // complexity appropriate for the environments within which it is employed. It is heavily 
   // configurable, has various operating modes and is suitable for a multitude of industrial 
   // applications.
   // 
   // IF YOU DON’T UNDERSTAND IT, DON’T USE IT. IF YOU DO USE IT, YOU DO SO AT YOUR OWN RISK.
   // 
   //                ━━━   ⬙⬙⬙⬙⬙⬙   ━━━
   // 
   // 
   // 
   // ▄▄▄▄▄▄▄▄▄▄▄▄▄▄▄▄▄▄▄▄▄▄▄▄▄▄▄▄▄▄▄▄▄▄▄▄▄▄▄▄▄▄▄▄
   // DOCUMENT REFERENCES
   // 
   //  ――――――――――――――――――――――――――――――――――――――――――
   //  REF.     DOCUMENT NO.       TITLE
   //  ――――――――――――――――――――――――――――――――――――――――――
   //  001  PS2001-5-0101-001   Quality Plan (QP)
   //  002  PS2001-5-0121-002   Validation Plan (VP)
   //  003  PS2001-5-0131-003   Test Plan (TP)
   //  004  PS2001-5-1101-001   User requirements specification (URS)
   //  005  PS2001-5-1111-001   Requirement Traceability Matrix (RTM)
   //  006  PS2001-5-2101-001   Functional Specification (FS) 
   //  007  PS2001-5-2211-001   Hardware Design Specification (HDS)
   //  008  PS2001-5-2311-001   Software Design Specification (SDS)
   //  009  PS2001-5-2313-011   Style Guide (SG)
   //  010  PS2001-5-234101-001    ES/WDP Configuration Manual
   //  011  PS2001-5-2312-fcNo.    Software Module Design Specification (SMDS)
   //  012  PS2001-5-2301-001   Software Module Register (SMR)
   //  013  PS2001-5-2302-011   Software Control and Mechanism (SCM)
   //  014  PS2001-5-7111-001   User Guide (UG)
   //  ――――――――――――――――――――――――――――――――――――――――――
   //  Note:   Where a block references another document not listed above (a calculation sheet
   //      for example), that document will be referenced separately in section 1.1 of the 
   //      block description for the block in question.
   // 
   // 
   // A full list of all project documentation is available here: 
   // 
   //      https://practicalseries.com/2001-pal/21-project/01-00-docs.html
   // 
   //                ━━━   ⬙⬙⬙⬙⬙⬙   ━━━
   // 
   // 
   // 
   // ▄▄▄▄▄▄▄▄▄▄▄▄▄▄▄▄▄▄▄▄▄▄▄▄▄▄▄▄▄▄▄▄▄▄▄▄▄▄▄▄▄▄▄▄
   // COMPLETED MODULES 
   // 
   //  ――――――――――――――――――――-―-- STATIC DATA       ― DYNAMIC  DAT A   ―
   //  BLOCK     NAME         REVISION    UDT/DB    REVISION  UDT/DB    REVISION  
   //  ――――――――――――――――――――――――――――――――――――――――――
   //  DB00801 St_ConstAiRawData  001.000   UT 00801   001.000       None
   //                  2024-05-16   DB00801   001.000       None
   //  ――――――――――――――――――――――――――――――――――――――――――
   //  DB00802 St_ConstAqRawData    001.000   UT 00802   001.000       None
   //                  2024-05-17   DB00802   001.000       None
   //  ――――――――――――――――――――――――――――――――――――――――――
   //  DB00851 St_ConstAiScaleData  001.000   UT 00851   001.000       None
   //                  2024-05-16   DB00851   001.000       None
   //  ――――――――――――――――――――――――――――――――――――――――――
   //  DB00851 St_ConstAqScaleData    001.000   UT 00852   001.000       None
   //                  2024-05-17   DB00852   001.000       None
   //  ――――――――――――――――――――――――――――――――――――――――――
   //  FC01001 StdSysGlobalData      002.000   None           UT 21000   002.000
   //                  2022-04-16                  UT 21001   002.000
   //                                    DB21001   002.000
   //  ――――――――――――――――――――――――――――――――――――――――――
   //  FC02001 StdInstAnalogRead    003.000   UT 02001   003.000    UT 22001   003.000
   //                  2024-05-16   DB02001   003.000       DB22001   003.000
   //  ――――――――――――――――――――――――――――――――――――――――――
   //  FC11001 StdDevValveIsol      002.000   UT 11001   002.000    UT 31001   002.000
   //                  2022-04-16   DB11001   002.000       DB31001   002.000
   //  ――――――――――――――――――――――――――――――――――――――――――
   //  FC11011 StdDevValve3Way      001.000   UT 11011   001.000    UT 31011   001.000
   //                  2022-06-11   DB11011   001.000       DB31011   001.000
   //  ――――――――――――――――――――――――――――――――――――――――――
   //  FC11101 StdDevValveBi      001.000   UT 11101   001.000    UT 31101   001.000
   //                  2023-02-02   DB11101   001.000       DB31101   001.000
   //  ――――――――――――――――――――――――――――――――――――――――――
   //  FC18001 StdSubScaleAI      003.000   None           None 
   //                  2022.08.31   None           None          
   //  ――――――――――――――――――――――――――――――――――――――――――
   //  FC18002 StdSubScaleAQ       001.000   None           None 
   //                  2022.09.01   None           None          
   //  ――――――――――――――――――――――――――――――――――――――――――
   //  FC18151 StdSubTimeEventRTC   002.000   None           UT 38151   002.000
   //                  2022-04-16   None           DB38151   002.000
   //  ――――――――――――――――――――――――――――――――――――――――――
   //  FC19511 StdDebugInst1Order    001.000   None           UT 39511   001.000
   //                  2023-03-03   None           DB39511   001.000
   //  ――――――――――――――――――――――――――――――――――――――――――
   //  FC19512 StdDebugInst2Order    002.000   None           UT 39512   002.000
   //                  2022-04-16   None           DB39512   002.000
   //  ――――――――――――――――――――――――――――――――――――――――――
   //  FC61000 DocGenExample     002.000   None           None 
   //                  2022-04-16   None           None          
   //  ――――――――――――――――――――――――――――――――――――――――――
   //  See Software Module Register [Ref. 012] for full details
   // 
   //                ━━━   ⬙⬙⬙⬙⬙⬙   ━━━
   // 
   // 
   // 
   // ▀▀▀▀▀▀▀▀▀▀▀▀▀▀▀▀▀▀▀▀▀▀▀▀▀▀▀▀▀▀▀▀▀▀▀▀▀▀▀▀▀▀▀▀
   // LICENCE AND CONTACT INFORMATION
   // 
   // This software and its associated documentation is made available under the MIT Licence:
   // 
   // ════════════════════════════════════════════
   // 
   // The MIT License (MIT)
   // 
   // Copyright © 2020 Michael Gledhill
   // 
   // Permission is hereby granted, free of charge, to any person obtaining a copy of this software 
   // and associated documentation files (the “Software”), to deal in the Software without restriction, 
   // including without limitation the rights to use, copy, modify, merge, publish, distribute, 
   // sublicense, and/or sell copies of the Software, and to permit persons to whom the Software is 
   // furnished to do so, subject to the following conditions: 
   // 
   // The above copyright notice and this permission notice shall be included in all copies or 
   // substantial portions of the Software.
   // 
   // THE SOFTWARE IS PROVIDED “AS IS”, WITHOUT WARRANTY OF ANY KIND, EXPRESS OR IMPLIED, 
   // INCLUDING BUT NOT LIMITED TO THE WARRANTIES OF MERCHANTABILITY, FITNESS FOR A 
   // PARTICULAR PURPOSE AND NON-INFRINGEMENT. IN NO EVENT SHALL THE AUTHORS OR COPYRIGHT 
   // HOLDERS BE LIABLE FOR ANY CLAIM, DAMAGES OR OTHER LIABILITY, WHETHER IN AN ACTION OF 
   // CONTRACT, TORT OR OTHERWISE, ARISING FROM, OUT OF OR IN CONNECTION WITH THE SOFTWARE 
   // OR THE USE OR OTHER DEALINGS IN THE SOFTWARE.
   // 
   // ════════════════════════════════════════════
   //                    ┌────────────┐
   // You can reach the author by email here:   │  mg@practicalseries.com  │
   //                    └────────────┘
   // Questions, corrections, constructive criticism and complaints (polite ones) are invited.
   // 
   // ▄▄▄▄▄▄▄▄▄▄▄▄▄▄▄▄▄▄▄▄▄▄▄▄▄▄▄▄▄▄▄▄▄▄▄▄▄▄▄▄▄▄▄▄
   // 
   //                ━━━   ⬙⬙⬙⬙⬙⬙   ━━━
   // 
   // 
   // 
   // ██████████████ █ █ █ █  END   █ █ █ █ ██████████████
END_REGION

REGION Network 2: Project revision and modification history
   // ▄▄▄▄▄▄▄▄▄▄▄▄▄▄▄▄▄▄▄▄▄▄▄▄▄▄▄▄▄▄▄▄▄▄▄▄▄▄▄▄▄▄▄▄
   // MODIFICATION HISTORY
   // 
   // The revision data herein contains the current revision of the whole software project 
   // (rather than of a particular block). The whole project is issued at a particular release and this is 
   // independent of individual module revisions.
   // 
   // The revision data shown here, in the network comments, contains additional information 
   // reflecting the software development workflow under the version control system (VCS) employed 
   // to track all software changes.
   // 
   // The VCS in use is the Git Source Code Management system in conjunction with the GitHub online 
   // hosting system. The software in its entirety is available in the GitHub remote repository:
   // 
   //      https://github.com/practicalseries/PS2001-pal-software
   // 
   // The repository is public and can be freely copied (forked in GitHub terminology) and used 
   // under the MIT licence. 
   // 
   // The MIT licence is reproduced in full in the last network of this software module.
   // 
   // 
   //  ———————————————————————————————————————————
   //  DATE       COMMIT TAG     AUTHOR        REASON FOR MODIFICATION
   //  ———————————————————————————————————————————
   //  2024.09.03    D0018      M. Gledhill      FC02001 — RELEASED FOR USE
   //                            FC18001 — RELEASED FOR USE
   //                            FC18002 — RELEASED FOR USE
   //                            DB00801, DB00802, DC00851 and
   //                            DB00852 all released for use
   // 
   //  2023.03.03    D0017      M. Gledhill      FC19511 — RELEASED FOR USE
   // 
   //  2023.02.02    D0016      M. Gledhill      FC11101 — RELEASED FOR USE
   // 
   //  2022.06.11    D0015      M. Gledhill      FC11011 — RELEASED FOR USE
   // 
   //  2022.05.03    D0014      M. Gledhill      Update to short URL links (now https)
   // 
   //  2022.04.16    D0011      M. Gledhill      All blocks — RE-RELEASED FOR USE
   //                            FC01001  FC02001  FC11001  FC18001 
   //                            FC18151  FC19152  FC61000
   // 
   //  2022.03.04    D0010      M. Gledhill      FC19512 — RELEASED FOR USE
   // 
   //  2021.08.23    D0009      M. Gledhill      FC11001 — RELEASED FOR USE
   // 
   //  2021.05.26    D0008      M. Gledhill      FC02001 — RELEASED FOR USE
   // 
   //  2021.05.22    D0007      M. Gledhill      FC18001 — RELEASED FOR USE
   // 
   //  2021.05.11    D0006      M. Gledhill      FC01001 — RELEASED FOR USE
   // 
   //  2021.05.02    D0005      M. Gledhill      Typographical corrections only
   // 
   //  2021.05.02    D0004      M. Gledhill      Typographical corrections only
   // 
   //  2021.02.19    D0003      M. Gledhill      FC18151 — RELEASED FOR USE
   // 
   //  2021.02.18    D0002      M. Gledhill      Baseline build
   // 
   //  2021.02.18    D0001      M. Gledhill      Hardware build
   // 
   //  2021.02.18    D0000      M. Gledhill      Initial commit — repository created
   //  ———————————————————————————————————————————
   // 
   // 
   // ▄▄▄▄▄▄▄▄▄▄▄▄▄▄▄▄▄▄▄▄▄▄▄▄▄▄▄▄▄▄▄▄▄▄▄▄▄▄▄▄▄▄▄▄
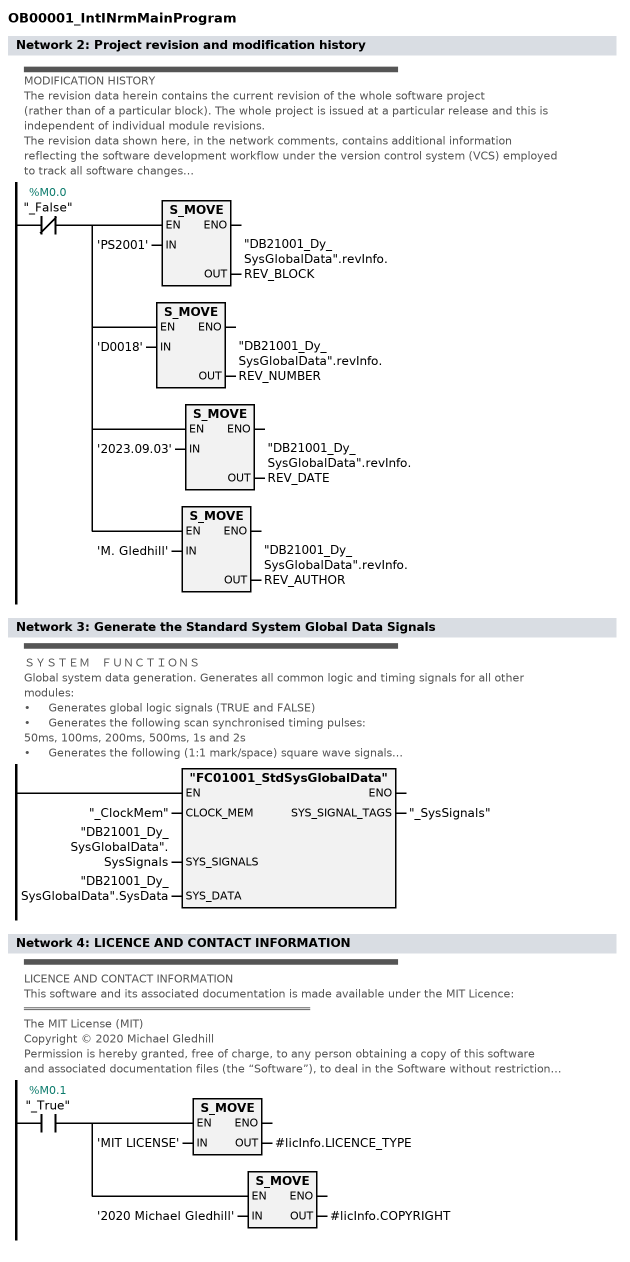
   RUNG wire#powerrail
      I_Contact( "_False" )
      wire#w1
      S_Move(in := 'PS2001', out => "DB21001_Dy_SysGlobalData".revInfo.REV_BLOCK)
   END_RUNG
   RUNG wire#w1
      S_Move(in := 'D0018', out => "DB21001_Dy_SysGlobalData".revInfo.REV_NUMBER)
   END_RUNG
   RUNG wire#w1
      S_Move(in := '2023.09.03', out => "DB21001_Dy_SysGlobalData".revInfo.REV_DATE)
   END_RUNG
   RUNG wire#w1
      S_Move(in := 'M. Gledhill', out => "DB21001_Dy_SysGlobalData".revInfo.REV_AUTHOR)
   END_RUNG
   // the same network as SCL:
   IF NOT "_False" THEN
       "DB21001_Dy_SysGlobalData".revInfo.REV_BLOCK := 'PS2001';
       "DB21001_Dy_SysGlobalData".revInfo.REV_NUMBER := 'D0018';
       "DB21001_Dy_SysGlobalData".revInfo.REV_DATE := '2023.09.03';
       "DB21001_Dy_SysGlobalData".revInfo.REV_AUTHOR := 'M. Gledhill';
   END_IF;
END_REGION

REGION Network 3: Generate the Standard System Global Data Signals
   // ▀▀▀▀▀▀▀▀▀▀▀▀▀▀▀▀▀▀▀▀▀▀▀▀▀▀▀▀▀▀▀▀▀▀▀▀▀▀▀▀▀▀▀▀
   // ＳＹＳＴＥＭ ＦＵＮＣＴＩＯＮＳ
   // 
   // Global system data generation. Generates all common logic and timing signals for all other 
   // modules:
   // 
   //    •   Generates global logic signals (TRUE and FALSE)
   // 
   //    •   Generates the following scan synchronised timing pulses:
   //        50ms, 100ms, 200ms, 500ms, 1s and 2s
   // 
   //    •   Generates the following (1:1 mark/space) square wave signals:
   //        100ms, 200ms, 500ms, 1s and 2s
   // 
   //    •   Generates odd and even (alternating) cycle tick-tock signals
   // 
   //    •   Generates a first-cycle signal indicating the controller has just started
   // 
   //    •   Records the cycle time of the last, maximum and minimum controller cycles
   // 
   //    •   Reads the controller internal real time clock and converts the values to discrete 
   //      integer values containing: year, month, day, day of week, hour, minute, second 
   //      and millisecond
   // 
   // The block must be the first non-debug block call within the main organisation block (OB 1).
   // ▄▄▄▄▄▄▄▄▄▄▄▄▄▄▄▄▄▄▄▄▄▄▄▄▄▄▄▄▄▄▄▄▄▄▄▄▄▄▄▄▄▄▄▄
   RUNG wire#powerrail
      "FC01001_StdSysGlobalData"(CLOCK_MEM := "_ClockMem", SYS_SIGNALS := "DB21001_Dy_SysGlobalData".SysSignals, SYS_DATA := "DB21001_Dy_SysGlobalData".SysData, SYS_SIGNAL_TAGS => "_SysSignals")
   END_RUNG
   // the same network as SCL:
   "FC01001_StdSysGlobalData"(CLOCK_MEM := "_ClockMem",
                           SYS_SIGNALS := "DB21001_Dy_SysGlobalData".SysSignals,
                           SYS_DATA := "DB21001_Dy_SysGlobalData".SysData,
                           SYS_SIGNAL_TAGS => "_SysSignals");
END_REGION

